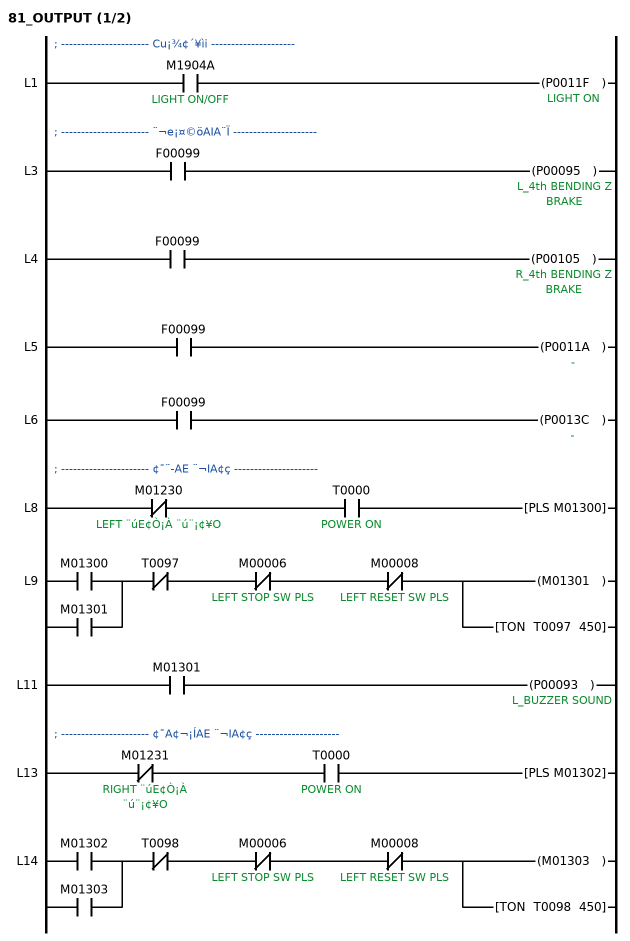
[picture p312: 81_OUTPUT rungs L1-L14]
// ---------------------- Cu¡¾¢´¥ìi ---------------------
; L1
LOAD      M1904A	// LIGHT ON/OFF
OUT       P0011F	// LIGHT ON
// ---------------------- ¨¬e¡¤©öAIA¨Ï ---------------------
; L3
LOAD      F00099
OUT       P00095	// L_4th BENDING Z BRAKE
; L4
LOAD      F00099
OUT       P00105	// R_4th BENDING Z BRAKE
; L5
LOAD      F00099
OUT       P0011A	// -
; L6
LOAD      F00099
OUT       P0013C	// -
// ---------------------- ¢¯¨­AE ¨¬IA¢ç ---------------------
; L8
LOAD NOT  M01230	// LEFT ¨úE¢Ò¡À ¨ú¨¡¢¥O
AND       T0000	// POWER ON
OUTP      M01300
; L9
LOAD      M01300
OR        M01301
AND NOT   T0097
AND NOT   M00006	// LEFT STOP SW PLS
AND NOT   M00008	// LEFT RESET SW PLS
OUT       M01301
TON       T0097 450
; L11
LOAD      M01301
OUT       P00093	// L_BUZZER SOUND
// ---------------------- ¢¯A¢¬¡ÍAE ¨¬IA¢ç ---------------------
; L13
LOAD NOT  M01231	// RIGHT ¨úE¢Ò¡À ¨ú¨¡¢¥O
AND       T0000	// POWER ON
OUTP      M01302
; L14
LOAD      M01302
OR        M01303
AND NOT   T0098
AND NOT   M00006	// LEFT STOP SW PLS
AND NOT   M00008	// LEFT RESET SW PLS
OUT       M01303
TON       T0098 450

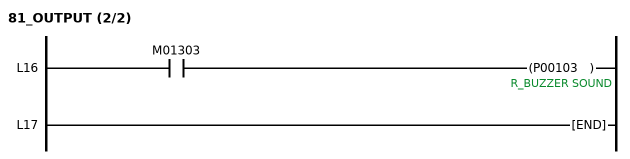
; L16
LOAD      M01303
OUT       P00103	// R_BUZZER SOUND
; L17
END

PROGRAM 82_L_MANUAL (task: ¨ö¨¬A¥ì CA¡¤I¡¾¡¿¡¤¡Í)

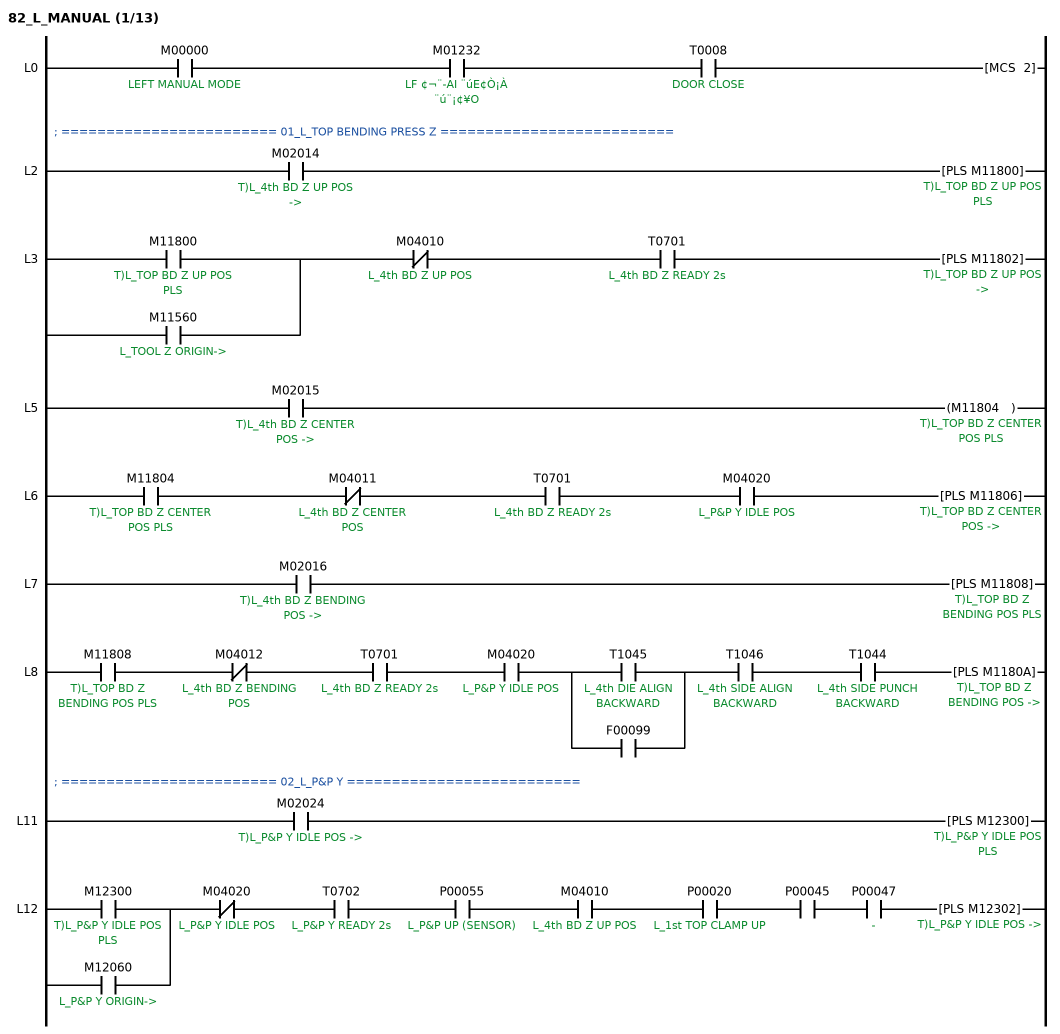
; L0
LOAD      M00000	// LEFT MANUAL MODE
AND       M01232	// LF ¢¬¨­AI ¨úE¢Ò¡À ¨ú¨¡¢¥O
AND       T0008	// DOOR CLOSE
MCS       2
// ======================== 01_L_TOP BENDING PRESS Z ==========================
; L2
LOAD      M02014	// T)L_4th BD Z UP POS ->
OUTP      M11800	// T)L_TOP BD Z UP POS PLS
; L3
LOAD      M11800	// T)L_TOP BD Z UP POS PLS
OR        M11560	// L_TOOL Z ORIGIN->
AND NOT   M04010	// L_4th BD Z UP POS
AND       T0701	// L_4th BD Z READY 2s
OUTP      M11802	// T)L_TOP BD Z UP POS ->
; L5
LOAD      M02015	// T)L_4th BD Z CENTER POS ->
OUT       M11804	// T)L_TOP BD Z CENTER POS PLS
; L6
LOAD      M11804	// T)L_TOP BD Z CENTER POS PLS
AND NOT   M04011	// L_4th BD Z CENTER POS
AND       T0701	// L_4th BD Z READY 2s
AND       M04020	// L_P&P Y IDLE POS
OUTP      M11806	// T)L_TOP BD Z CENTER POS ->
; L7
LOAD      M02016	// T)L_4th BD Z BENDING POS ->
OUTP      M11808	// T)L_TOP BD Z BENDING POS PLS
; L8
LOAD      M11808	// T)L_TOP BD Z BENDING POS PLS
AND NOT   M04012	// L_4th BD Z BENDING POS
AND       T0701	// L_4th BD Z READY 2s
AND       M04020	// L_P&P Y IDLE POS
LOAD      T1045	// L_4th DIE ALIGN BACKWARD
OR        F00099
AND LOAD
AND       T1046	// L_4th SIDE ALIGN BACKWARD
AND       T1044	// L_4th SIDE PUNCH BACKWARD
OUTP      M1180A	// T)L_TOP BD Z BENDING POS ->
// ======================== 02_L_P&P Y ==========================
; L11
LOAD      M02024	// T)L_P&P Y IDLE POS ->
OUTP      M12300	// T)L_P&P Y IDLE POS PLS
; L12
LOAD      M12300	// T)L_P&P Y IDLE POS PLS
OR        M12060	// L_P&P Y ORIGIN->
AND NOT   M04020	// L_P&P Y IDLE POS
AND       T0702	// L_P&P Y READY 2s
AND       P00055	// L_P&P UP (SENSOR)
AND       M04010	// L_4th BD Z UP POS
AND       P00020	// L_1st TOP CLAMP UP
AND       P00045
AND       P00047	// -
OUTP      M12302	// T)L_P&P Y IDLE POS ->

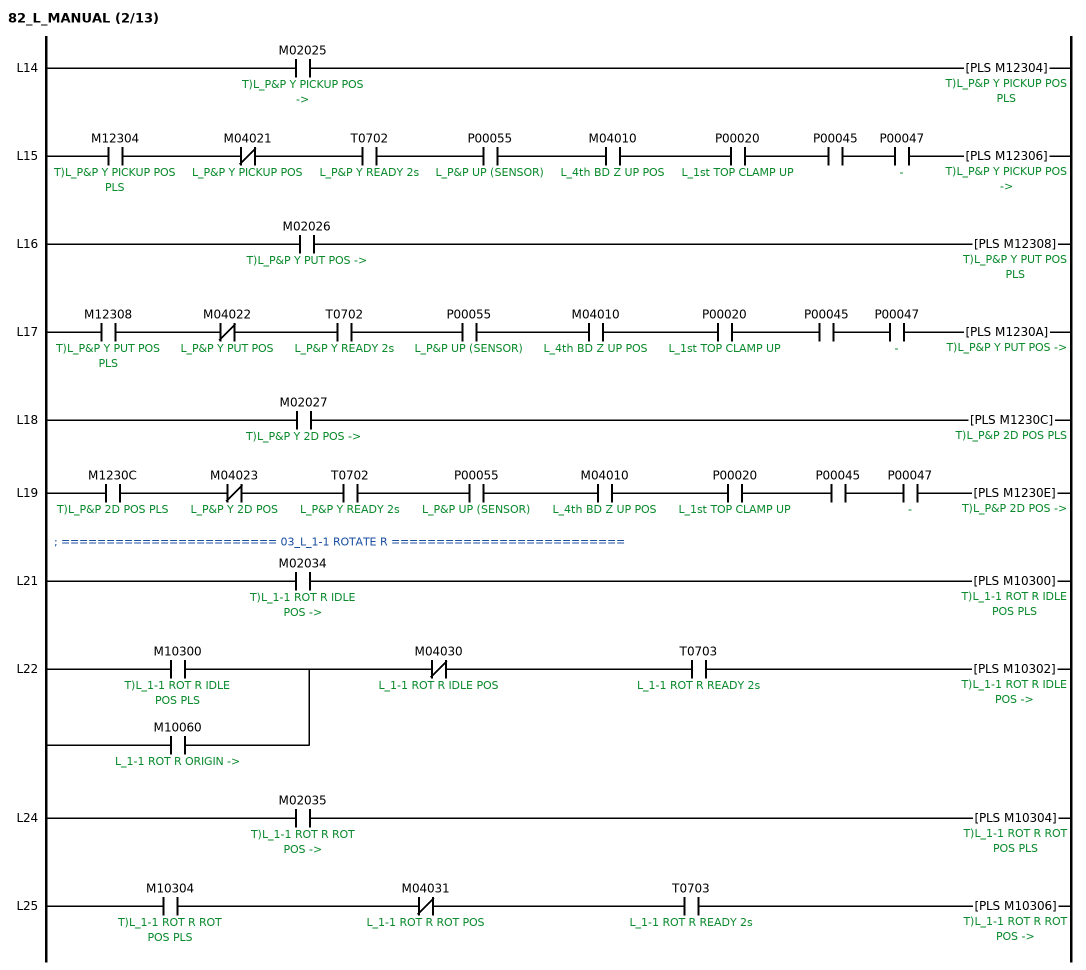
; L14
LOAD      M02025	// T)L_P&P Y PICKUP POS ->
OUTP      M12304	// T)L_P&P Y PICKUP POS PLS
; L15
LOAD      M12304	// T)L_P&P Y PICKUP POS PLS
AND NOT   M04021	// L_P&P Y PICKUP POS
AND       T0702	// L_P&P Y READY 2s
AND       P00055	// L_P&P UP (SENSOR)
AND       M04010	// L_4th BD Z UP POS
AND       P00020	// L_1st TOP CLAMP UP
AND       P00045
AND       P00047	// -
OUTP      M12306	// T)L_P&P Y PICKUP POS ->
; L16
LOAD      M02026	// T)L_P&P Y PUT POS ->
OUTP      M12308	// T)L_P&P Y PUT POS PLS
; L17
LOAD      M12308	// T)L_P&P Y PUT POS PLS
AND NOT   M04022	// L_P&P Y PUT POS
AND       T0702	// L_P&P Y READY 2s
AND       P00055	// L_P&P UP (SENSOR)
AND       M04010	// L_4th BD Z UP POS
AND       P00020	// L_1st TOP CLAMP UP
AND       P00045
AND       P00047	// -
OUTP      M1230A	// T)L_P&P Y PUT POS ->
; L18
LOAD      M02027	// T)L_P&P Y 2D POS ->
OUTP      M1230C	// T)L_P&P 2D POS PLS
; L19
LOAD      M1230C	// T)L_P&P 2D POS PLS
AND NOT   M04023	// L_P&P Y 2D POS
AND       T0702	// L_P&P Y READY 2s
AND       P00055	// L_P&P UP (SENSOR)
AND       M04010	// L_4th BD Z UP POS
AND       P00020	// L_1st TOP CLAMP UP
AND       P00045
AND       P00047	// -
OUTP      M1230E	// T)L_P&P 2D POS ->
// ======================== 03_L_1-1 ROTATE R ==========================
; L21
LOAD      M02034	// T)L_1-1 ROT R IDLE POS ->
OUTP      M10300	// T)L_1-1 ROT R IDLE POS PLS
; L22
LOAD      M10300	// T)L_1-1 ROT R IDLE POS PLS
OR        M10060	// L_1-1 ROT R ORIGIN ->
AND NOT   M04030	// L_1-1 ROT R IDLE POS
AND       T0703	// L_1-1 ROT R READY 2s
OUTP      M10302	// T)L_1-1 ROT R IDLE POS ->
; L24
LOAD      M02035	// T)L_1-1 ROT R ROT POS ->
OUTP      M10304	// T)L_1-1 ROT R ROT POS PLS
; L25
LOAD      M10304	// T)L_1-1 ROT R ROT POS PLS
AND NOT   M04031	// L_1-1 ROT R ROT POS
AND       T0703	// L_1-1 ROT R READY 2s
OUTP      M10306	// T)L_1-1 ROT R ROT POS ->

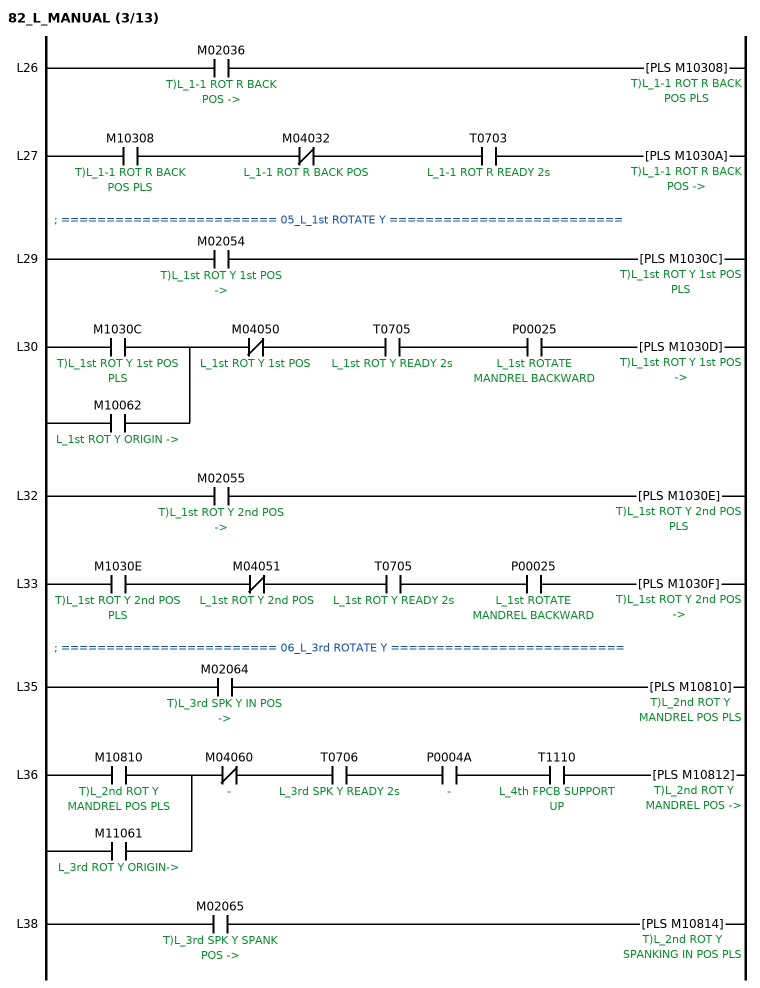
; L26
LOAD      M02036	// T)L_1-1 ROT R BACK POS ->
OUTP      M10308	// T)L_1-1 ROT R BACK POS PLS
; L27
LOAD      M10308	// T)L_1-1 ROT R BACK POS PLS
AND NOT   M04032	// L_1-1 ROT R BACK POS
AND       T0703	// L_1-1 ROT R READY 2s
OUTP      M1030A	// T)L_1-1 ROT R BACK POS ->
// ======================== 05_L_1st ROTATE Y ==========================
; L29
LOAD      M02054	// T)L_1st ROT Y 1st POS ->
OUTP      M1030C	// T)L_1st ROT Y 1st POS PLS
; L30
LOAD      M1030C	// T)L_1st ROT Y 1st POS PLS
OR        M10062	// L_1st ROT Y ORIGIN ->
AND NOT   M04050	// L_1st ROT Y 1st POS
AND       T0705	// L_1st ROT Y READY 2s
AND       P00025	// L_1st ROTATE MANDREL BACKWARD
OUTP      M1030D	// T)L_1st ROT Y 1st POS ->
; L32
LOAD      M02055	// T)L_1st ROT Y 2nd POS ->
OUTP      M1030E	// T)L_1st ROT Y 2nd POS PLS
; L33
LOAD      M1030E	// T)L_1st ROT Y 2nd POS PLS
AND NOT   M04051	// L_1st ROT Y 2nd POS
AND       T0705	// L_1st ROT Y READY 2s
AND       P00025	// L_1st ROTATE MANDREL BACKWARD
OUTP      M1030F	// T)L_1st ROT Y 2nd POS ->
// ======================== 06_L_3rd ROTATE Y ==========================
; L35
LOAD      M02064	// T)L_3rd SPK Y IN POS ->
OUTP      M10810	// T)L_2nd ROT Y MANDREL POS PLS
; L36
LOAD      M10810	// T)L_2nd ROT Y MANDREL POS PLS
OR        M11061	// L_3rd ROT Y ORIGIN->
AND NOT   M04060	// -
AND       T0706	// L_3rd SPK Y READY 2s
AND       P0004A	// -
AND       T1110	// L_4th FPCB SUPPORT UP
OUTP      M10812	// T)L_2nd ROT Y MANDREL POS ->
; L38
LOAD      M02065	// T)L_3rd SPK Y SPANK POS ->
OUTP      M10814	// T)L_2nd ROT Y SPANKING IN POS PLS

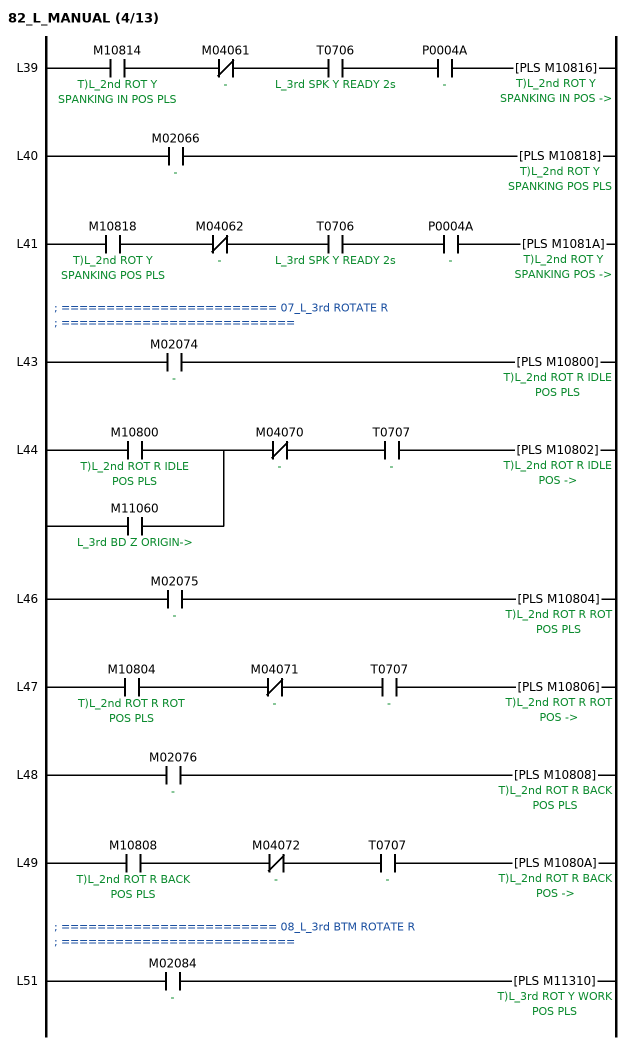
; L39
LOAD      M10814	// T)L_2nd ROT Y SPANKING IN POS PLS
AND NOT   M04061	// -
AND       T0706	// L_3rd SPK Y READY 2s
AND       P0004A	// -
OUTP      M10816	// T)L_2nd ROT Y SPANKING IN POS ->
; L40
LOAD      M02066	// -
OUTP      M10818	// T)L_2nd ROT Y SPANKING POS PLS
; L41
LOAD      M10818	// T)L_2nd ROT Y SPANKING POS PLS
AND NOT   M04062	// -
AND       T0706	// L_3rd SPK Y READY 2s
AND       P0004A	// -
OUTP      M1081A	// T)L_2nd ROT Y SPANKING POS ->
// ======================== 07_L_3rd ROTATE R ==========================
; L43
LOAD      M02074	// -
OUTP      M10800	// T)L_2nd ROT R IDLE POS PLS
; L44
LOAD      M10800	// T)L_2nd ROT R IDLE POS PLS
OR        M11060	// L_3rd BD Z ORIGIN->
AND NOT   M04070	// -
AND       T0707	// -
OUTP      M10802	// T)L_2nd ROT R IDLE POS ->
; L46
LOAD      M02075	// -
OUTP      M10804	// T)L_2nd ROT R ROT POS PLS
; L47
LOAD      M10804	// T)L_2nd ROT R ROT POS PLS
AND NOT   M04071	// -
AND       T0707	// -
OUTP      M10806	// T)L_2nd ROT R ROT POS ->
; L48
LOAD      M02076	// -
OUTP      M10808	// T)L_2nd ROT R BACK POS PLS
; L49
LOAD      M10808	// T)L_2nd ROT R BACK POS PLS
AND NOT   M04072	// -
AND       T0707	// -
OUTP      M1080A	// T)L_2nd ROT R BACK POS ->
// ======================== 08_L_3rd BTM ROTATE R ==========================
; L51
LOAD      M02084	// -
OUTP      M11310	// T)L_3rd ROT Y WORK POS PLS

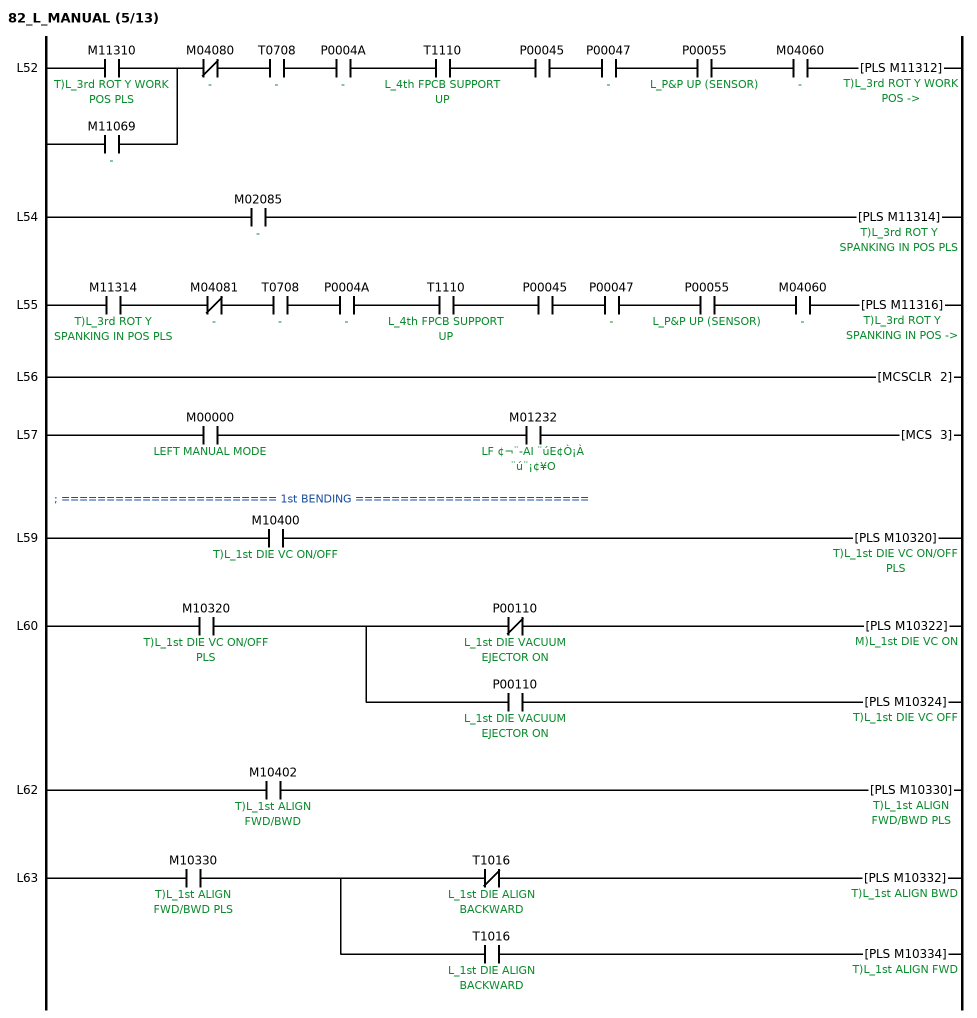
; L52
LOAD      M11310	// T)L_3rd ROT Y WORK POS PLS
OR        M11069	// -
AND NOT   M04080	// -
AND       T0708	// -
AND       P0004A	// -
AND       T1110	// L_4th FPCB SUPPORT UP
AND       P00045
AND       P00047	// -
AND       P00055	// L_P&P UP (SENSOR)
AND       M04060	// -
OUTP      M11312	// T)L_3rd ROT Y WORK POS ->
; L54
LOAD      M02085	// -
OUTP      M11314	// T)L_3rd ROT Y SPANKING IN POS PLS
; L55
LOAD      M11314	// T)L_3rd ROT Y SPANKING IN POS PLS
AND NOT   M04081	// -
AND       T0708	// -
AND       P0004A	// -
AND       T1110	// L_4th FPCB SUPPORT UP
AND       P00045
AND       P00047	// -
AND       P00055	// L_P&P UP (SENSOR)
AND       M04060	// -
OUTP      M11316	// T)L_3rd ROT Y SPANKING IN POS ->
; L56
MCSCLR    2
; L57
LOAD      M00000	// LEFT MANUAL MODE
AND       M01232	// LF ¢¬¨­AI ¨úE¢Ò¡À ¨ú¨¡¢¥O
MCS       3
// ======================== 1st BENDING ==========================
; L59
LOAD      M10400	// T)L_1st DIE VC ON/OFF
OUTP      M10320	// T)L_1st DIE VC ON/OFF PLS
; L60
LOAD      M10320	// T)L_1st DIE VC ON/OFF PLS
MPUSH
AND NOT   P00110	// L_1st DIE VACUUM EJECTOR ON
OUTP      M10322	// M)L_1st DIE VC ON
MPOP
AND       P00110	// L_1st DIE VACUUM EJECTOR ON
OUTP      M10324	// T)L_1st DIE VC OFF
; L62
LOAD      M10402	// T)L_1st ALIGN FWD/BWD
OUTP      M10330	// T)L_1st ALIGN FWD/BWD PLS
; L63
LOAD      M10330	// T)L_1st ALIGN FWD/BWD PLS
MPUSH
AND NOT   T1016	// L_1st DIE ALIGN BACKWARD
OUTP      M10332	// T)L_1st ALIGN BWD
MPOP
AND       T1016	// L_1st DIE ALIGN BACKWARD
OUTP      M10334	// T)L_1st ALIGN FWD

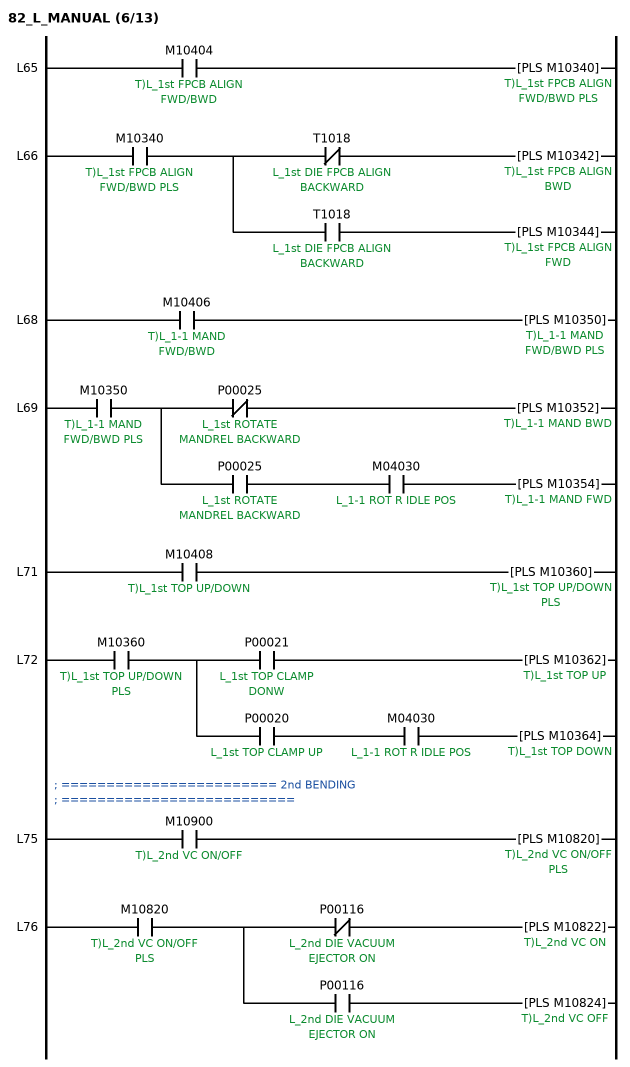
; L65
LOAD      M10404	// T)L_1st FPCB ALIGN FWD/BWD
OUTP      M10340	// T)L_1st FPCB ALIGN FWD/BWD PLS
; L66
LOAD      M10340	// T)L_1st FPCB ALIGN FWD/BWD PLS
MPUSH
AND NOT   T1018	// L_1st DIE FPCB ALIGN BACKWARD
OUTP      M10342	// T)L_1st FPCB ALIGN BWD
MPOP
AND       T1018	// L_1st DIE FPCB ALIGN BACKWARD
OUTP      M10344	// T)L_1st FPCB ALIGN FWD
; L68
LOAD      M10406	// T)L_1-1 MAND FWD/BWD
OUTP      M10350	// T)L_1-1 MAND FWD/BWD PLS
; L69
LOAD      M10350	// T)L_1-1 MAND FWD/BWD PLS
MPUSH
AND NOT   P00025	// L_1st ROTATE MANDREL BACKWARD
OUTP      M10352	// T)L_1-1 MAND BWD
MPOP
AND       P00025	// L_1st ROTATE MANDREL BACKWARD
AND       M04030	// L_1-1 ROT R IDLE POS
OUTP      M10354	// T)L_1-1 MAND FWD
; L71
LOAD      M10408	// T)L_1st TOP UP/DOWN
OUTP      M10360	// T)L_1st TOP UP/DOWN PLS
; L72
LOAD      M10360	// T)L_1st TOP UP/DOWN PLS
MPUSH
AND       P00021	// L_1st TOP CLAMP DONW
OUTP      M10362	// T)L_1st TOP UP
MPOP
AND       P00020	// L_1st TOP CLAMP UP
AND       M04030	// L_1-1 ROT R IDLE POS
OUTP      M10364	// T)L_1st TOP DOWN
// ======================== 2nd BENDING ==========================
; L75
LOAD      M10900	// T)L_2nd VC ON/OFF
OUTP      M10820	// T)L_2nd VC ON/OFF PLS
; L76
LOAD      M10820	// T)L_2nd VC ON/OFF PLS
MPUSH
AND NOT   P00116	// L_2nd DIE VACUUM EJECTOR ON
OUTP      M10822	// T)L_2nd VC ON
MPOP
AND       P00116	// L_2nd DIE VACUUM EJECTOR ON
OUTP      M10824	// T)L_2nd VC OFF

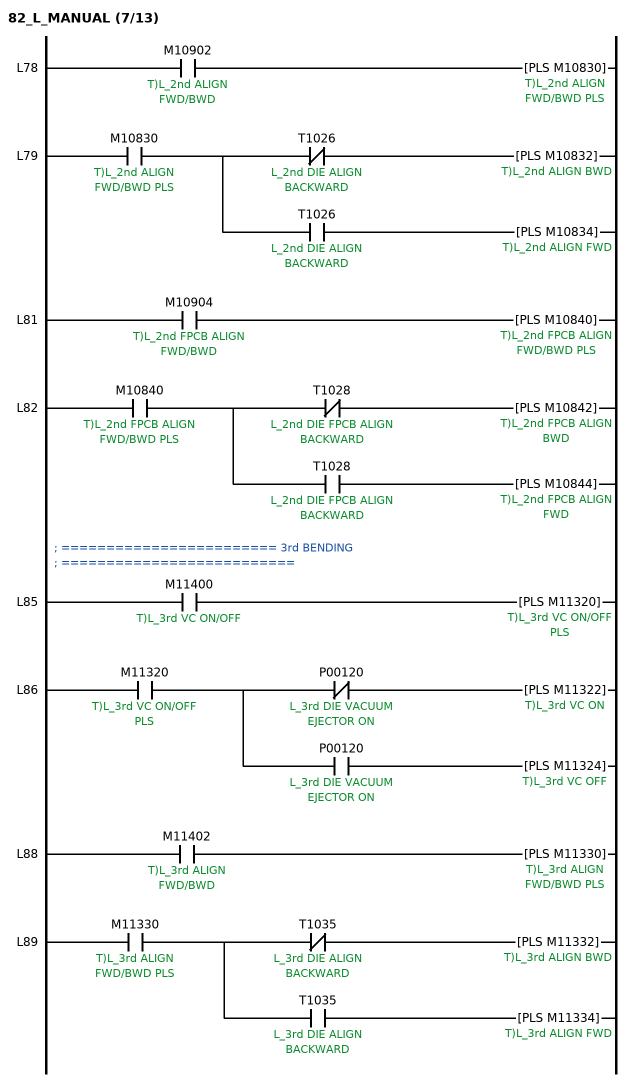
; L78
LOAD      M10902	// T)L_2nd ALIGN FWD/BWD
OUTP      M10830	// T)L_2nd ALIGN FWD/BWD PLS
; L79
LOAD      M10830	// T)L_2nd ALIGN FWD/BWD PLS
MPUSH
AND NOT   T1026	// L_2nd DIE ALIGN BACKWARD
OUTP      M10832	// T)L_2nd ALIGN BWD
MPOP
AND       T1026	// L_2nd DIE ALIGN BACKWARD
OUTP      M10834	// T)L_2nd ALIGN FWD
; L81
LOAD      M10904	// T)L_2nd FPCB ALIGN FWD/BWD
OUTP      M10840	// T)L_2nd FPCB ALIGN FWD/BWD PLS
; L82
LOAD      M10840	// T)L_2nd FPCB ALIGN FWD/BWD PLS
MPUSH
AND NOT   T1028	// L_2nd DIE FPCB ALIGN BACKWARD
OUTP      M10842	// T)L_2nd FPCB ALIGN BWD
MPOP
AND       T1028	// L_2nd DIE FPCB ALIGN BACKWARD
OUTP      M10844	// T)L_2nd FPCB ALIGN FWD
// ======================== 3rd BENDING ==========================
; L85
LOAD      M11400	// T)L_3rd VC ON/OFF
OUTP      M11320	// T)L_3rd VC ON/OFF PLS
; L86
LOAD      M11320	// T)L_3rd VC ON/OFF PLS
MPUSH
AND NOT   P00120	// L_3rd DIE VACUUM EJECTOR ON
OUTP      M11322	// T)L_3rd VC ON
MPOP
AND       P00120	// L_3rd DIE VACUUM EJECTOR ON
OUTP      M11324	// T)L_3rd VC OFF
; L88
LOAD      M11402	// T)L_3rd ALIGN FWD/BWD
OUTP      M11330	// T)L_3rd ALIGN FWD/BWD PLS
; L89
LOAD      M11330	// T)L_3rd ALIGN FWD/BWD PLS
MPUSH
AND NOT   T1035	// L_3rd DIE ALIGN BACKWARD
OUTP      M11332	// T)L_3rd ALIGN BWD
MPOP
AND       T1035	// L_3rd DIE ALIGN BACKWARD
OUTP      M11334	// T)L_3rd ALIGN FWD

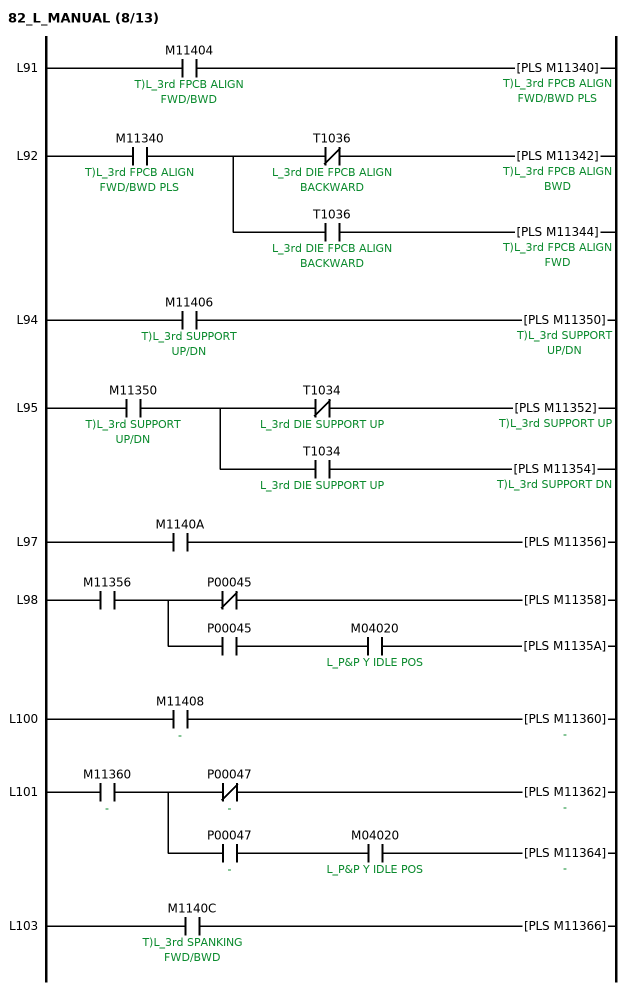
; L91
LOAD      M11404	// T)L_3rd FPCB ALIGN FWD/BWD
OUTP      M11340	// T)L_3rd FPCB ALIGN FWD/BWD PLS
; L92
LOAD      M11340	// T)L_3rd FPCB ALIGN FWD/BWD PLS
MPUSH
AND NOT   T1036	// L_3rd DIE FPCB ALIGN BACKWARD
OUTP      M11342	// T)L_3rd FPCB ALIGN BWD
MPOP
AND       T1036	// L_3rd DIE FPCB ALIGN BACKWARD
OUTP      M11344	// T)L_3rd FPCB ALIGN FWD
; L94
LOAD      M11406	// T)L_3rd SUPPORT UP/DN
OUTP      M11350	// T)L_3rd SUPPORT UP/DN
; L95
LOAD      M11350	// T)L_3rd SUPPORT UP/DN
MPUSH
AND NOT   T1034	// L_3rd DIE SUPPORT UP
OUTP      M11352	// T)L_3rd SUPPORT UP
MPOP
AND       T1034	// L_3rd DIE SUPPORT UP
OUTP      M11354	// T)L_3rd SUPPORT DN
; L97
LOAD      M1140A
OUTP      M11356
; L98
LOAD      M11356
MPUSH
AND NOT   P00045
OUTP      M11358
MPOP
AND       P00045
AND       M04020	// L_P&P Y IDLE POS
OUTP      M1135A
; L100
LOAD      M11408	// -
OUTP      M11360	// -
; L101
LOAD      M11360	// -
MPUSH
AND NOT   P00047	// -
OUTP      M11362	// -
MPOP
AND       P00047	// -
AND       M04020	// L_P&P Y IDLE POS
OUTP      M11364	// -
; L103
LOAD      M1140C	// T)L_3rd SPANKING FWD/BWD
OUTP      M11366

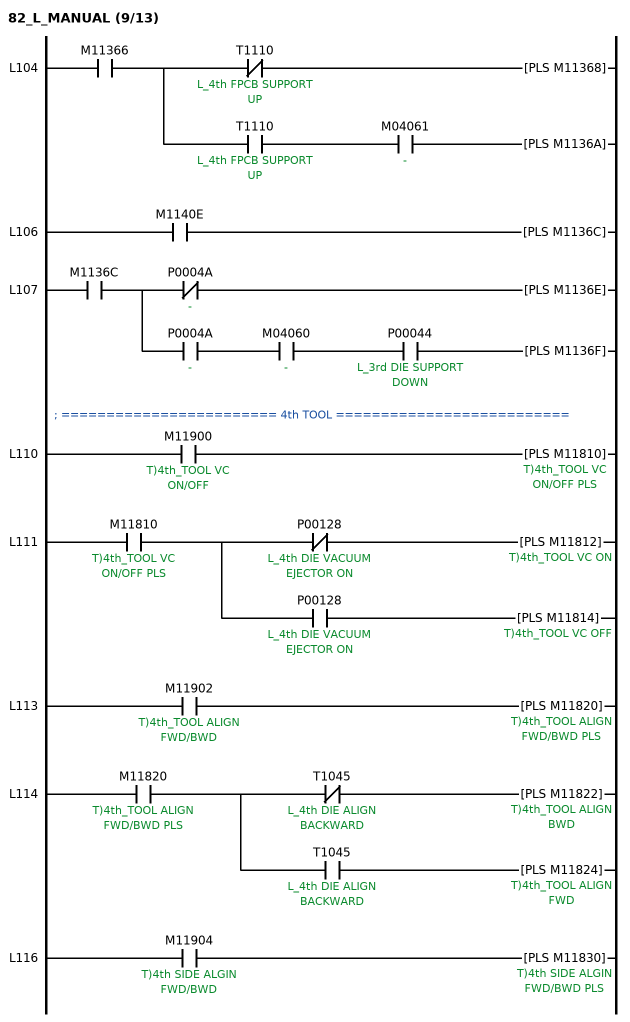
; L104
LOAD      M11366
MPUSH
AND NOT   T1110	// L_4th FPCB SUPPORT UP
OUTP      M11368
MPOP
AND       T1110	// L_4th FPCB SUPPORT UP
AND       M04061	// -
OUTP      M1136A
; L106
LOAD      M1140E
OUTP      M1136C
; L107
LOAD      M1136C
MPUSH
AND NOT   P0004A	// -
OUTP      M1136E
MPOP
AND       P0004A	// -
AND       M04060	// -
AND       P00044	// L_3rd DIE SUPPORT DOWN
OUTP      M1136F
// ======================== 4th TOOL ==========================
; L110
LOAD      M11900	// T)4th_TOOL VC ON/OFF
OUTP      M11810	// T)4th_TOOL VC ON/OFF PLS
; L111
LOAD      M11810	// T)4th_TOOL VC ON/OFF PLS
MPUSH
AND NOT   P00128	// L_4th DIE VACUUM EJECTOR ON
OUTP      M11812	// T)4th_TOOL VC ON
MPOP
AND       P00128	// L_4th DIE VACUUM EJECTOR ON
OUTP      M11814	// T)4th_TOOL VC OFF
; L113
LOAD      M11902	// T)4th_TOOL ALIGN FWD/BWD
OUTP      M11820	// T)4th_TOOL ALIGN FWD/BWD PLS
; L114
LOAD      M11820	// T)4th_TOOL ALIGN FWD/BWD PLS
MPUSH
AND NOT   T1045	// L_4th DIE ALIGN BACKWARD
OUTP      M11822	// T)4th_TOOL ALIGN BWD
MPOP
AND       T1045	// L_4th DIE ALIGN BACKWARD
OUTP      M11824	// T)4th_TOOL ALIGN FWD
; L116
LOAD      M11904	// T)4th SIDE ALGIN FWD/BWD
OUTP      M11830	// T)4th SIDE ALGIN FWD/BWD PLS

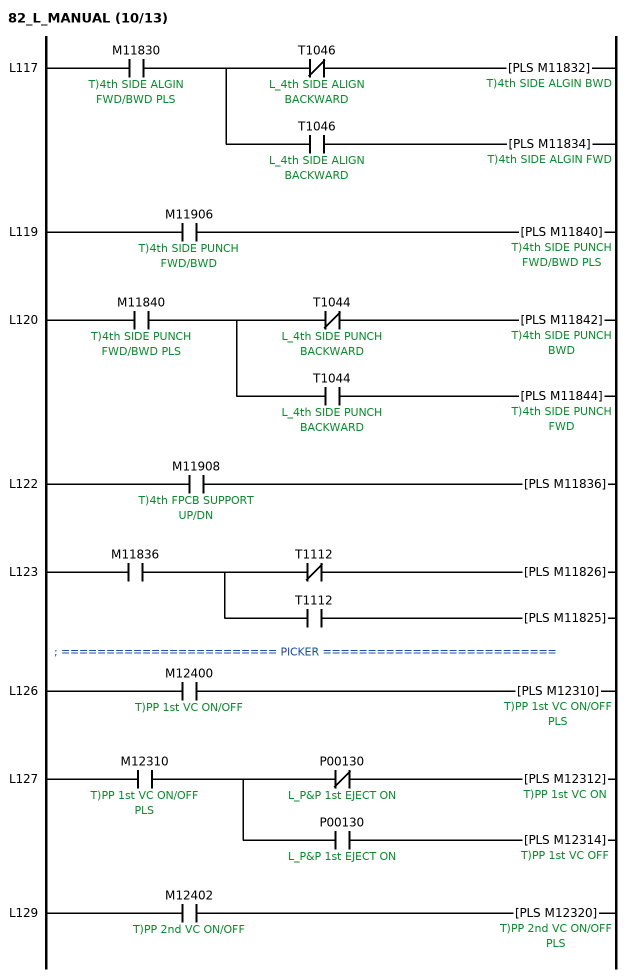
; L117
LOAD      M11830	// T)4th SIDE ALGIN FWD/BWD PLS
MPUSH
AND NOT   T1046	// L_4th SIDE ALIGN BACKWARD
OUTP      M11832	// T)4th SIDE ALGIN BWD
MPOP
AND       T1046	// L_4th SIDE ALIGN BACKWARD
OUTP      M11834	// T)4th SIDE ALGIN FWD
; L119
LOAD      M11906	// T)4th SIDE PUNCH FWD/BWD
OUTP      M11840	// T)4th SIDE PUNCH FWD/BWD PLS
; L120
LOAD      M11840	// T)4th SIDE PUNCH FWD/BWD PLS
MPUSH
AND NOT   T1044	// L_4th SIDE PUNCH BACKWARD
OUTP      M11842	// T)4th SIDE PUNCH BWD
MPOP
AND       T1044	// L_4th SIDE PUNCH BACKWARD
OUTP      M11844	// T)4th SIDE PUNCH FWD
; L122
LOAD      M11908	// T)4th FPCB SUPPORT UP/DN
OUTP      M11836
; L123
LOAD      M11836
MPUSH
AND NOT   T1112
OUTP      M11826
MPOP
AND       T1112
OUTP      M11825
// ======================== PICKER ==========================
; L126
LOAD      M12400	// T)PP 1st VC ON/OFF
OUTP      M12310	// T)PP 1st VC ON/OFF PLS
; L127
LOAD      M12310	// T)PP 1st VC ON/OFF PLS
MPUSH
AND NOT   P00130	// L_P&P 1st EJECT ON
OUTP      M12312	// T)PP 1st VC ON
MPOP
AND       P00130	// L_P&P 1st EJECT ON
OUTP      M12314	// T)PP 1st VC OFF
; L129
LOAD      M12402	// T)PP 2nd VC ON/OFF
OUTP      M12320	// T)PP 2nd VC ON/OFF PLS

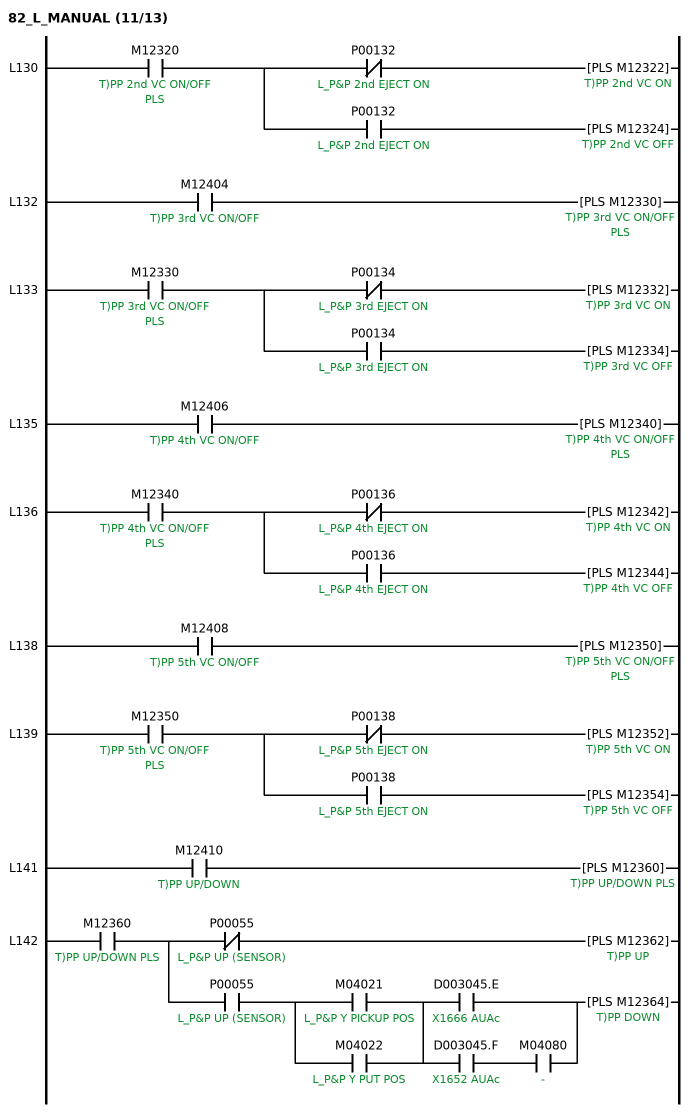
; L130
LOAD      M12320	// T)PP 2nd VC ON/OFF PLS
MPUSH
AND NOT   P00132	// L_P&P 2nd EJECT ON
OUTP      M12322	// T)PP 2nd VC ON
MPOP
AND       P00132	// L_P&P 2nd EJECT ON
OUTP      M12324	// T)PP 2nd VC OFF
; L132
LOAD      M12404	// T)PP 3rd VC ON/OFF
OUTP      M12330	// T)PP 3rd VC ON/OFF PLS
; L133
LOAD      M12330	// T)PP 3rd VC ON/OFF PLS
MPUSH
AND NOT   P00134	// L_P&P 3rd EJECT ON
OUTP      M12332	// T)PP 3rd VC ON
MPOP
AND       P00134	// L_P&P 3rd EJECT ON
OUTP      M12334	// T)PP 3rd VC OFF
; L135
LOAD      M12406	// T)PP 4th VC ON/OFF
OUTP      M12340	// T)PP 4th VC ON/OFF PLS
; L136
LOAD      M12340	// T)PP 4th VC ON/OFF PLS
MPUSH
AND NOT   P00136	// L_P&P 4th EJECT ON
OUTP      M12342	// T)PP 4th VC ON
MPOP
AND       P00136	// L_P&P 4th EJECT ON
OUTP      M12344	// T)PP 4th VC OFF
; L138
LOAD      M12408	// T)PP 5th VC ON/OFF
OUTP      M12350	// T)PP 5th VC ON/OFF PLS
; L139
LOAD      M12350	// T)PP 5th VC ON/OFF PLS
MPUSH
AND NOT   P00138	// L_P&P 5th EJECT ON
OUTP      M12352	// T)PP 5th VC ON
MPOP
AND       P00138	// L_P&P 5th EJECT ON
OUTP      M12354	// T)PP 5th VC OFF
; L141
LOAD      M12410	// T)PP UP/DOWN
OUTP      M12360	// T)PP UP/DOWN PLS
; L142
LOAD      M12360	// T)PP UP/DOWN PLS
MPUSH
AND NOT   P00055	// L_P&P UP (SENSOR)
OUTP      M12362	// T)PP UP
MPOP
AND       P00055	// L_P&P UP (SENSOR)
LOAD      M04021	// L_P&P Y PICKUP POS
OR        M04022	// L_P&P Y PUT POS
AND LOAD
LOAD      D003045.E	// X1666 AUAc
LOAD      D003045.F	// X1652 AUAc
AND       M04080	// -
OR LOAD
AND LOAD
OUTP      M12364	// T)PP DOWN

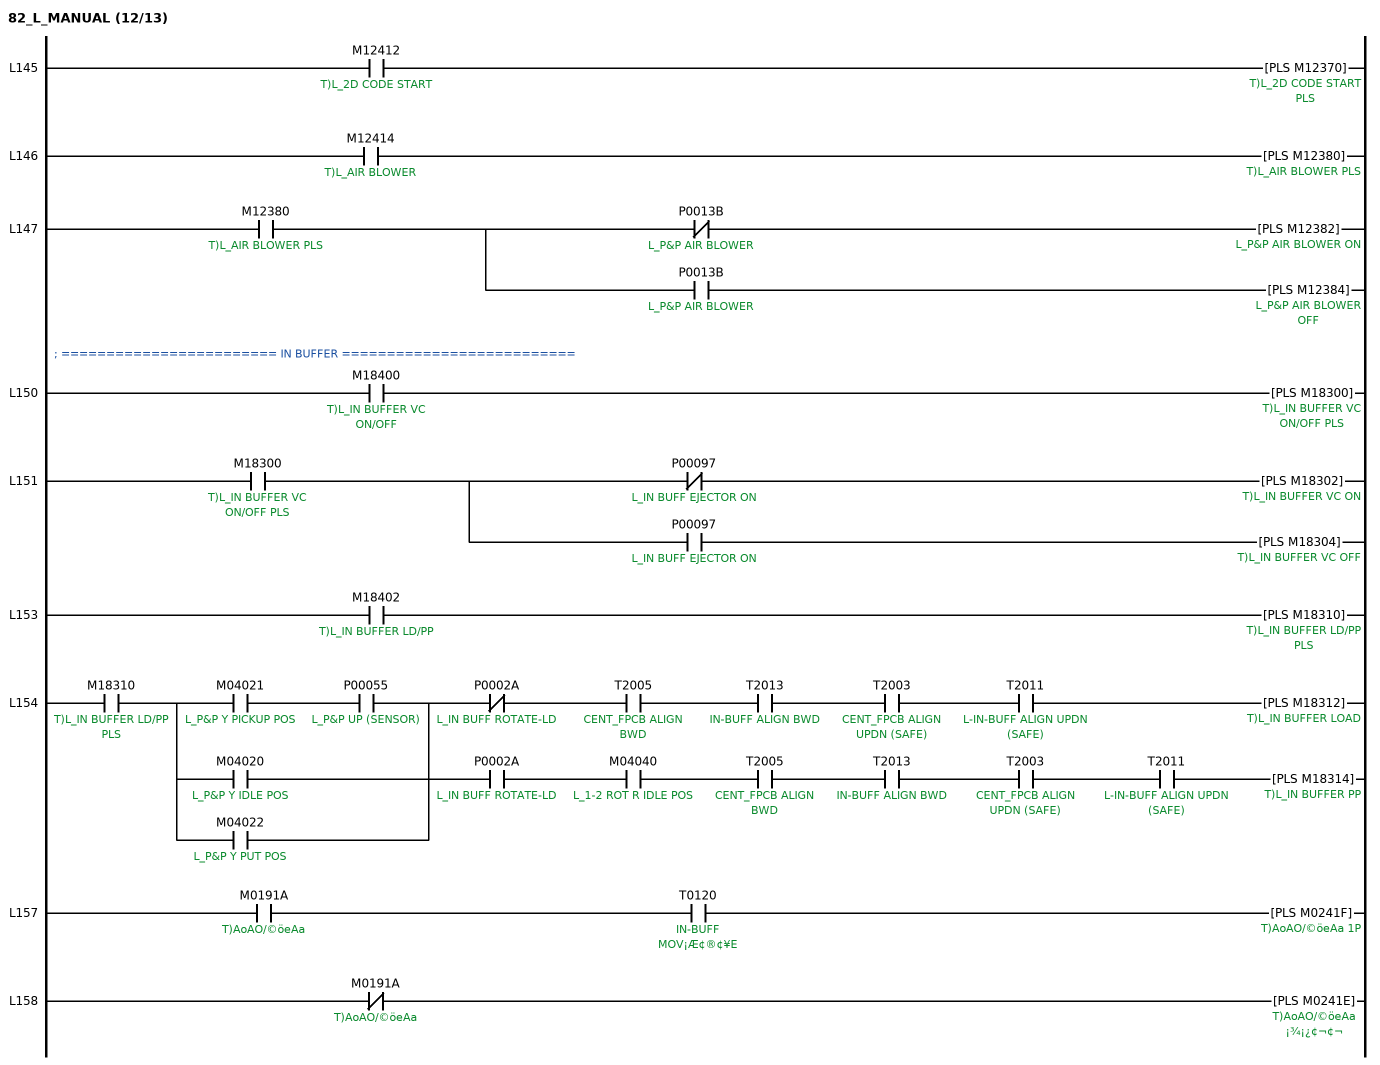
; L145
LOAD      M12412	// T)L_2D CODE START
OUTP      M12370	// T)L_2D CODE START PLS
; L146
LOAD      M12414	// T)L_AIR BLOWER
OUTP      M12380	// T)L_AIR BLOWER PLS
; L147
LOAD      M12380	// T)L_AIR BLOWER PLS
MPUSH
AND NOT   P0013B	// L_P&P AIR BLOWER
OUTP      M12382	// L_P&P AIR BLOWER ON
MPOP
AND       P0013B	// L_P&P AIR BLOWER
OUTP      M12384	// L_P&P AIR BLOWER OFF
// ======================== IN BUFFER ==========================
; L150
LOAD      M18400	// T)L_IN BUFFER VC ON/OFF
OUTP      M18300	// T)L_IN BUFFER VC ON/OFF PLS
; L151
LOAD      M18300	// T)L_IN BUFFER VC ON/OFF PLS
MPUSH
AND NOT   P00097	// L_IN BUFF EJECTOR ON
OUTP      M18302	// T)L_IN BUFFER VC ON
MPOP
AND       P00097	// L_IN BUFF EJECTOR ON
OUTP      M18304	// T)L_IN BUFFER VC OFF
; L153
LOAD      M18402	// T)L_IN BUFFER LD/PP
OUTP      M18310	// T)L_IN BUFFER LD/PP PLS
; L154
LOAD      M18310	// T)L_IN BUFFER LD/PP PLS
LOAD      M04021	// L_P&P Y PICKUP POS
AND       P00055	// L_P&P UP (SENSOR)
OR        M04020	// L_P&P Y IDLE POS
OR        M04022	// L_P&P Y PUT POS
AND LOAD
MPUSH
AND NOT   P0002A	// L_IN BUFF ROTATE-LD
AND       T2005	// CENT_FPCB ALIGN BWD
AND       T2013	// IN-BUFF ALIGN BWD
AND       T2003	// CENT_FPCB ALIGN UPDN (SAFE)
AND       T2011	// L-IN-BUFF ALIGN UPDN (SAFE)
OUTP      M18312	// T)L_IN BUFFER LOAD
MPOP
AND       P0002A	// L_IN BUFF ROTATE-LD
AND       M04040	// L_1-2 ROT R IDLE POS
AND       T2005	// CENT_FPCB ALIGN BWD
AND       T2013	// IN-BUFF ALIGN BWD
AND       T2003	// CENT_FPCB ALIGN UPDN (SAFE)
AND       T2011	// L-IN-BUFF ALIGN UPDN (SAFE)
OUTP      M18314	// T)L_IN BUFFER PP
; L157
LOAD      M0191A	// T)AoAO/©öeAa
AND       T0120	// IN-BUFF MOV¡Æ¢®¢¥E
OUTP      M0241F	// T)AoAO/©öeAa 1P
; L158
LOAD NOT  M0191A	// T)AoAO/©öeAa
OUTP      M0241E	// T)AoAO/©öeAa ¡¾¡¿¢¬¢¬

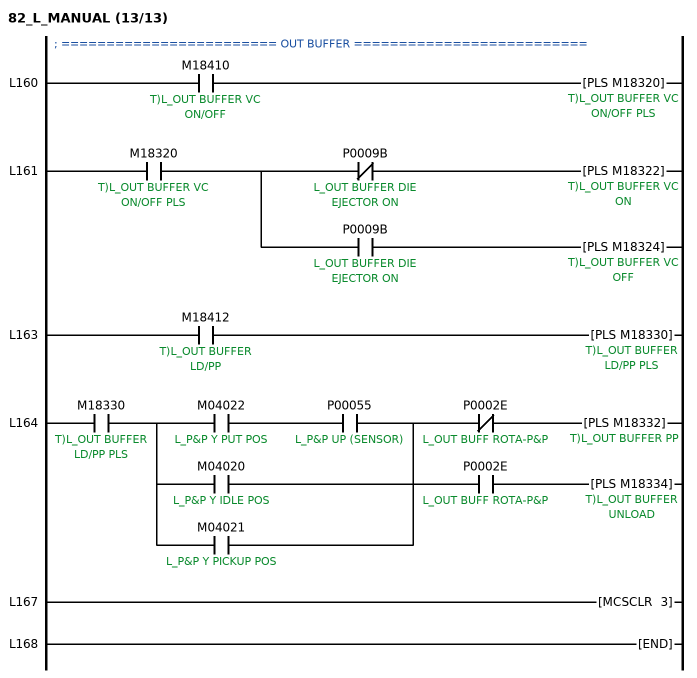
// ======================== OUT BUFFER ==========================
; L160
LOAD      M18410	// T)L_OUT BUFFER VC ON/OFF
OUTP      M18320	// T)L_OUT BUFFER VC ON/OFF PLS
; L161
LOAD      M18320	// T)L_OUT BUFFER VC ON/OFF PLS
MPUSH
AND NOT   P0009B	// L_OUT BUFFER DIE EJECTOR ON
OUTP      M18322	// T)L_OUT BUFFER VC ON
MPOP
AND       P0009B	// L_OUT BUFFER DIE EJECTOR ON
OUTP      M18324	// T)L_OUT BUFFER VC OFF
; L163
LOAD      M18412	// T)L_OUT BUFFER LD/PP
OUTP      M18330	// T)L_OUT BUFFER LD/PP PLS
; L164
LOAD      M18330	// T)L_OUT BUFFER LD/PP PLS
LOAD      M04022	// L_P&P Y PUT POS
AND       P00055	// L_P&P UP (SENSOR)
OR        M04020	// L_P&P Y IDLE POS
OR        M04021	// L_P&P Y PICKUP POS
AND LOAD
MPUSH
AND NOT   P0002E	// L_OUT BUFF ROTA-P&P
OUTP      M18332	// T)L_OUT BUFFER PP
MPOP
AND       P0002E	// L_OUT BUFF ROTA-P&P
OUTP      M18334	// T)L_OUT BUFFER UNLOAD
; L167
MCSCLR    3
; L168
END

PROGRAM 83_R_MANUAL (task: ¨ö¨¬A¥ì CA¡¤I¡¾¡¿¡¤¡Í)

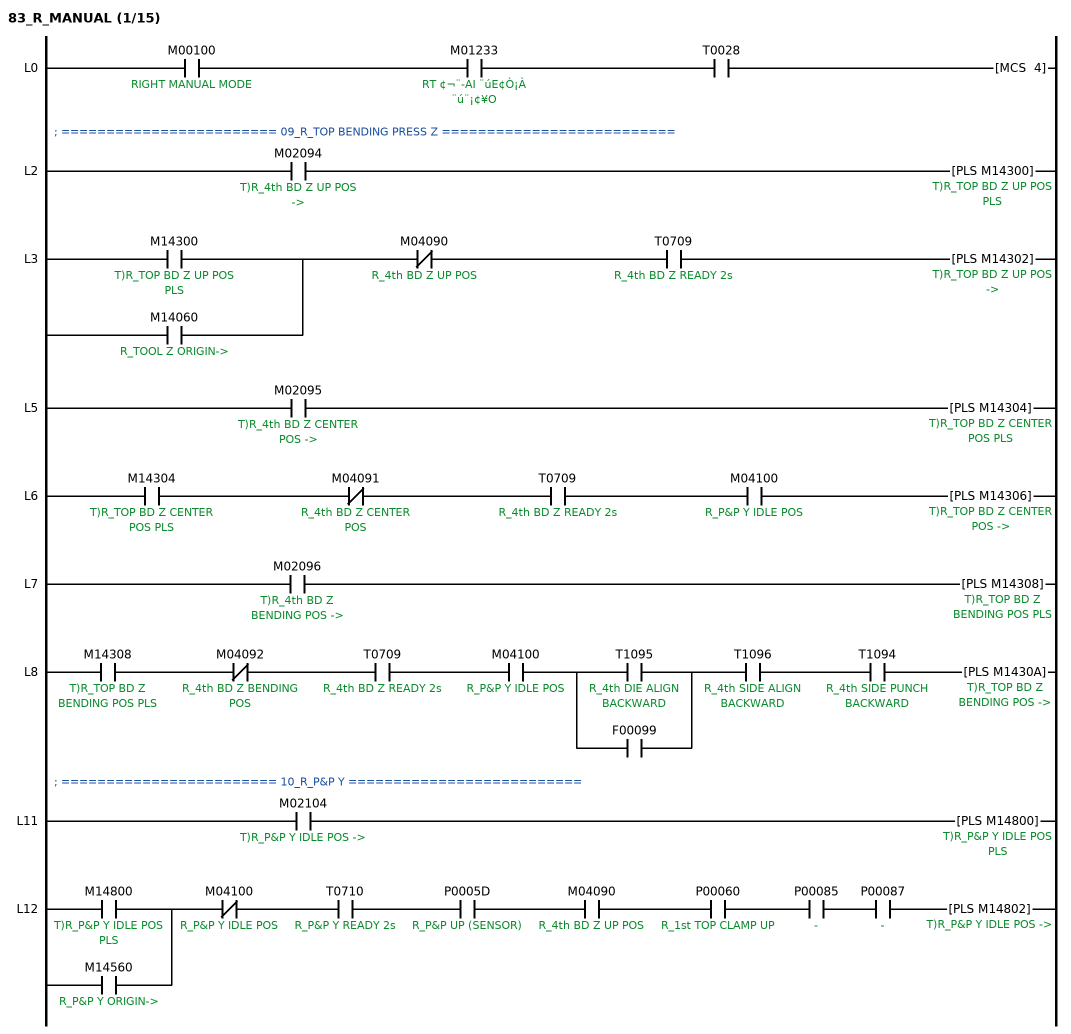
; L0
LOAD      M00100	// RIGHT MANUAL MODE
AND       M01233	// RT ¢¬¨­AI ¨úE¢Ò¡À ¨ú¨¡¢¥O
AND       T0028
MCS       4
// ======================== 09_R_TOP BENDING PRESS Z ==========================
; L2
LOAD      M02094	// T)R_4th BD Z UP POS ->
OUTP      M14300	// T)R_TOP BD Z UP POS PLS
; L3
LOAD      M14300	// T)R_TOP BD Z UP POS PLS
OR        M14060	// R_TOOL Z ORIGIN->
AND NOT   M04090	// R_4th BD Z UP POS
AND       T0709	// R_4th BD Z READY 2s
OUTP      M14302	// T)R_TOP BD Z UP POS ->
; L5
LOAD      M02095	// T)R_4th BD Z CENTER POS ->
OUTP      M14304	// T)R_TOP BD Z CENTER POS PLS
; L6
LOAD      M14304	// T)R_TOP BD Z CENTER POS PLS
AND NOT   M04091	// R_4th BD Z CENTER POS
AND       T0709	// R_4th BD Z READY 2s
AND       M04100	// R_P&P Y IDLE POS
OUTP      M14306	// T)R_TOP BD Z CENTER POS ->
; L7
LOAD      M02096	// T)R_4th BD Z BENDING POS ->
OUTP      M14308	// T)R_TOP BD Z BENDING POS PLS
; L8
LOAD      M14308	// T)R_TOP BD Z BENDING POS PLS
AND NOT   M04092	// R_4th BD Z BENDING POS
AND       T0709	// R_4th BD Z READY 2s
AND       M04100	// R_P&P Y IDLE POS
LOAD      T1095	// R_4th DIE ALIGN BACKWARD
OR        F00099
AND LOAD
AND       T1096	// R_4th SIDE ALIGN BACKWARD
AND       T1094	// R_4th SIDE PUNCH BACKWARD
OUTP      M1430A	// T)R_TOP BD Z BENDING POS ->
// ======================== 10_R_P&P Y ==========================
; L11
LOAD      M02104	// T)R_P&P Y IDLE POS ->
OUTP      M14800	// T)R_P&P Y IDLE POS PLS
; L12
LOAD      M14800	// T)R_P&P Y IDLE POS PLS
OR        M14560	// R_P&P Y ORIGIN->
AND NOT   M04100	// R_P&P Y IDLE POS
AND       T0710	// R_P&P Y READY 2s
AND       P0005D	// R_P&P UP (SENSOR)
AND       M04090	// R_4th BD Z UP POS
AND       P00060	// R_1st TOP CLAMP UP
AND       P00085	// -
AND       P00087	// -
OUTP      M14802	// T)R_P&P Y IDLE POS ->

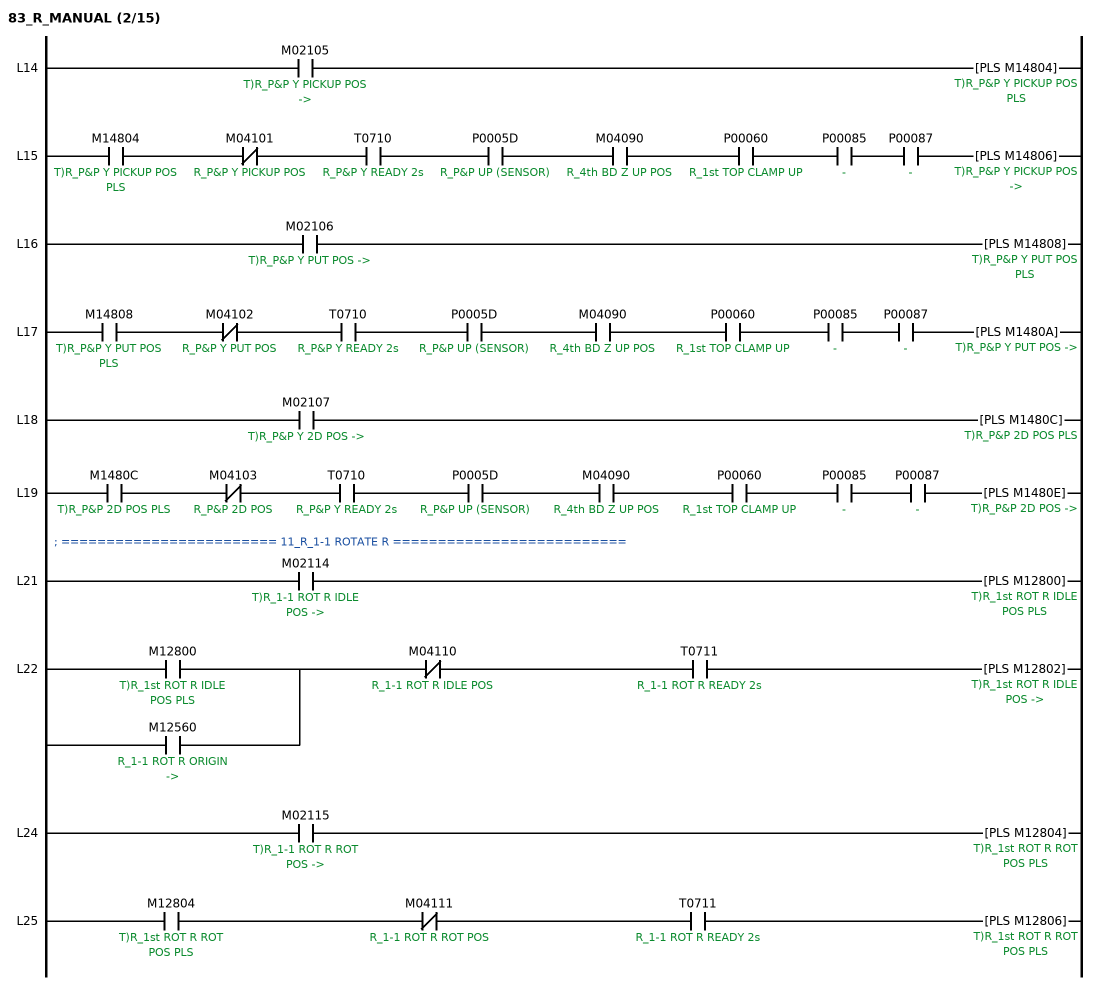
; L14
LOAD      M02105	// T)R_P&P Y PICKUP POS ->
OUTP      M14804	// T)R_P&P Y PICKUP POS PLS
; L15
LOAD      M14804	// T)R_P&P Y PICKUP POS PLS
AND NOT   M04101	// R_P&P Y PICKUP POS
AND       T0710	// R_P&P Y READY 2s
AND       P0005D	// R_P&P UP (SENSOR)
AND       M04090	// R_4th BD Z UP POS
AND       P00060	// R_1st TOP CLAMP UP
AND       P00085	// -
AND       P00087	// -
OUTP      M14806	// T)R_P&P Y PICKUP POS ->
; L16
LOAD      M02106	// T)R_P&P Y PUT POS ->
OUTP      M14808	// T)R_P&P Y PUT POS PLS
; L17
LOAD      M14808	// T)R_P&P Y PUT POS PLS
AND NOT   M04102	// R_P&P Y PUT POS
AND       T0710	// R_P&P Y READY 2s
AND       P0005D	// R_P&P UP (SENSOR)
AND       M04090	// R_4th BD Z UP POS
AND       P00060	// R_1st TOP CLAMP UP
AND       P00085	// -
AND       P00087	// -
OUTP      M1480A	// T)R_P&P Y PUT POS ->
; L18
LOAD      M02107	// T)R_P&P Y 2D POS ->
OUTP      M1480C	// T)R_P&P 2D POS PLS
; L19
LOAD      M1480C	// T)R_P&P 2D POS PLS
AND NOT   M04103	// R_P&P 2D POS
AND       T0710	// R_P&P Y READY 2s
AND       P0005D	// R_P&P UP (SENSOR)
AND       M04090	// R_4th BD Z UP POS
AND       P00060	// R_1st TOP CLAMP UP
AND       P00085	// -
AND       P00087	// -
OUTP      M1480E	// T)R_P&P 2D POS ->
// ======================== 11_R_1-1 ROTATE R ==========================
; L21
LOAD      M02114	// T)R_1-1 ROT R IDLE POS ->
OUTP      M12800	// T)R_1st ROT R IDLE POS PLS
; L22
LOAD      M12800	// T)R_1st ROT R IDLE POS PLS
OR        M12560	// R_1-1 ROT R ORIGIN ->
AND NOT   M04110	// R_1-1 ROT R IDLE POS
AND       T0711	// R_1-1 ROT R READY 2s
OUTP      M12802	// T)R_1st ROT R IDLE POS ->
; L24
LOAD      M02115	// T)R_1-1 ROT R ROT POS ->
OUTP      M12804	// T)R_1st ROT R ROT POS PLS
; L25
LOAD      M12804	// T)R_1st ROT R ROT POS PLS
AND NOT   M04111	// R_1-1 ROT R ROT POS
AND       T0711	// R_1-1 ROT R READY 2s
OUTP      M12806	// T)R_1st ROT R ROT POS PLS

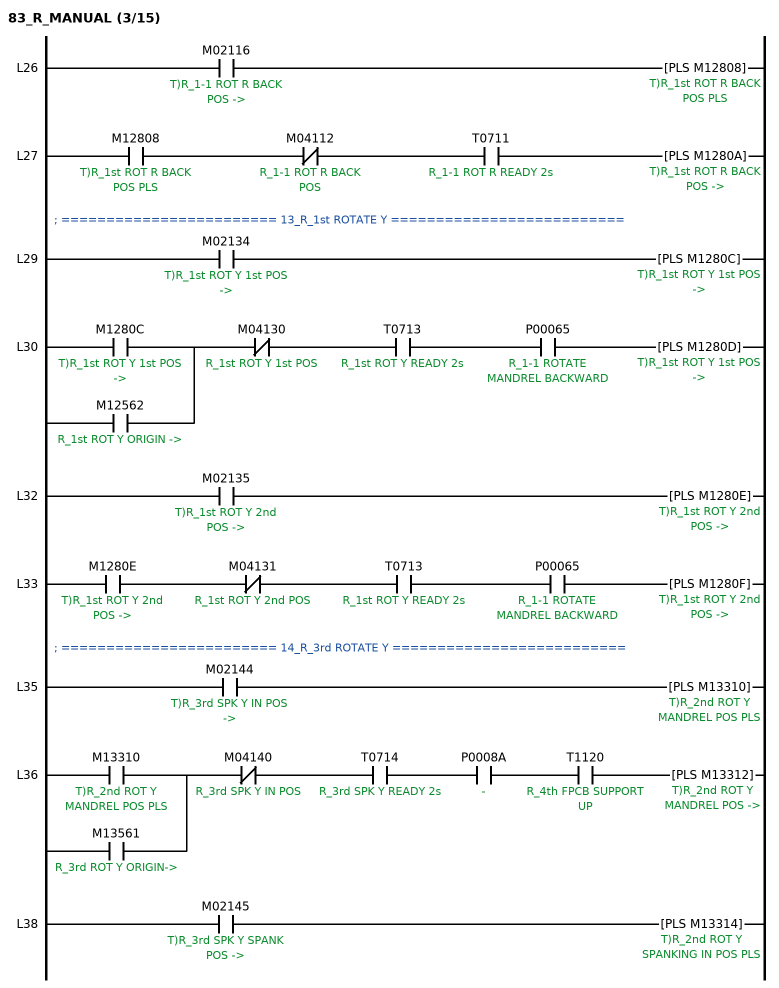
; L26
LOAD      M02116	// T)R_1-1 ROT R BACK POS ->
OUTP      M12808	// T)R_1st ROT R BACK POS PLS
; L27
LOAD      M12808	// T)R_1st ROT R BACK POS PLS
AND NOT   M04112	// R_1-1 ROT R BACK POS
AND       T0711	// R_1-1 ROT R READY 2s
OUTP      M1280A	// T)R_1st ROT R BACK POS ->
// ======================== 13_R_1st ROTATE Y ==========================
; L29
LOAD      M02134	// T)R_1st ROT Y 1st POS ->
OUTP      M1280C	// T)R_1st ROT Y 1st POS ->
; L30
LOAD      M1280C	// T)R_1st ROT Y 1st POS ->
OR        M12562	// R_1st ROT Y ORIGIN ->
AND NOT   M04130	// R_1st ROT Y 1st POS
AND       T0713	// R_1st ROT Y READY 2s
AND       P00065	// R_1-1 ROTATE MANDREL BACKWARD
OUTP      M1280D	// T)R_1st ROT Y 1st POS ->
; L32
LOAD      M02135	// T)R_1st ROT Y 2nd POS ->
OUTP      M1280E	// T)R_1st ROT Y 2nd POS ->
; L33
LOAD      M1280E	// T)R_1st ROT Y 2nd POS ->
AND NOT   M04131	// R_1st ROT Y 2nd POS
AND       T0713	// R_1st ROT Y READY 2s
AND       P00065	// R_1-1 ROTATE MANDREL BACKWARD
OUTP      M1280F	// T)R_1st ROT Y 2nd POS ->
// ======================== 14_R_3rd ROTATE Y ==========================
; L35
LOAD      M02144	// T)R_3rd SPK Y IN POS ->
OUTP      M13310	// T)R_2nd ROT Y MANDREL POS PLS
; L36
LOAD      M13310	// T)R_2nd ROT Y MANDREL POS PLS
OR        M13561	// R_3rd ROT Y ORIGIN->
AND NOT   M04140	// R_3rd SPK Y IN POS
AND       T0714	// R_3rd SPK Y READY 2s
AND       P0008A	// -
AND       T1120	// R_4th FPCB SUPPORT UP
OUTP      M13312	// T)R_2nd ROT Y MANDREL POS ->
; L38
LOAD      M02145	// T)R_3rd SPK Y SPANK POS ->
OUTP      M13314	// T)R_2nd ROT Y SPANKING IN POS PLS

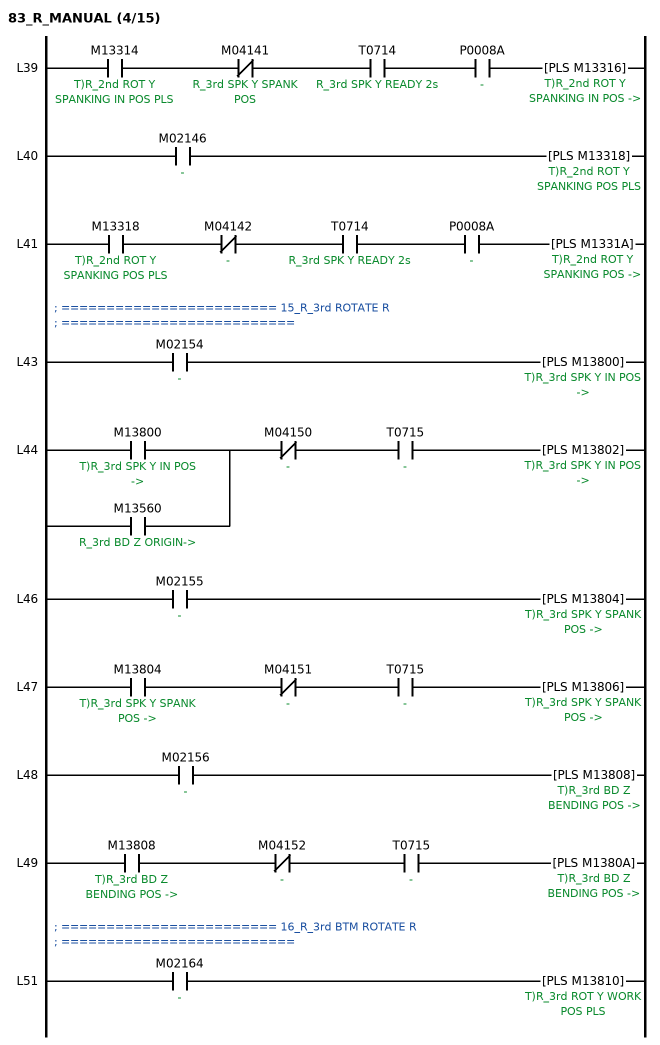
; L39
LOAD      M13314	// T)R_2nd ROT Y SPANKING IN POS PLS
AND NOT   M04141	// R_3rd SPK Y SPANK POS
AND       T0714	// R_3rd SPK Y READY 2s
AND       P0008A	// -
OUTP      M13316	// T)R_2nd ROT Y SPANKING IN POS ->
; L40
LOAD      M02146	// -
OUTP      M13318	// T)R_2nd ROT Y SPANKING POS PLS
; L41
LOAD      M13318	// T)R_2nd ROT Y SPANKING POS PLS
AND NOT   M04142	// -
AND       T0714	// R_3rd SPK Y READY 2s
AND       P0008A	// -
OUTP      M1331A	// T)R_2nd ROT Y SPANKING POS ->
// ======================== 15_R_3rd ROTATE R ==========================
; L43
LOAD      M02154	// -
OUTP      M13800	// T)R_3rd SPK Y IN POS ->
; L44
LOAD      M13800	// T)R_3rd SPK Y IN POS ->
OR        M13560	// R_3rd BD Z ORIGIN->
AND NOT   M04150	// -
AND       T0715	// -
OUTP      M13802	// T)R_3rd SPK Y IN POS ->
; L46
LOAD      M02155	// -
OUTP      M13804	// T)R_3rd SPK Y SPANK POS ->
; L47
LOAD      M13804	// T)R_3rd SPK Y SPANK POS ->
AND NOT   M04151	// -
AND       T0715	// -
OUTP      M13806	// T)R_3rd SPK Y SPANK POS ->
; L48
LOAD      M02156	// -
OUTP      M13808	// T)R_3rd BD Z BENDING POS ->
; L49
LOAD      M13808	// T)R_3rd BD Z BENDING POS ->
AND NOT   M04152	// -
AND       T0715	// -
OUTP      M1380A	// T)R_3rd BD Z BENDING POS ->
// ======================== 16_R_3rd BTM ROTATE R ==========================
; L51
LOAD      M02164	// -
OUTP      M13810	// T)R_3rd ROT Y WORK POS PLS

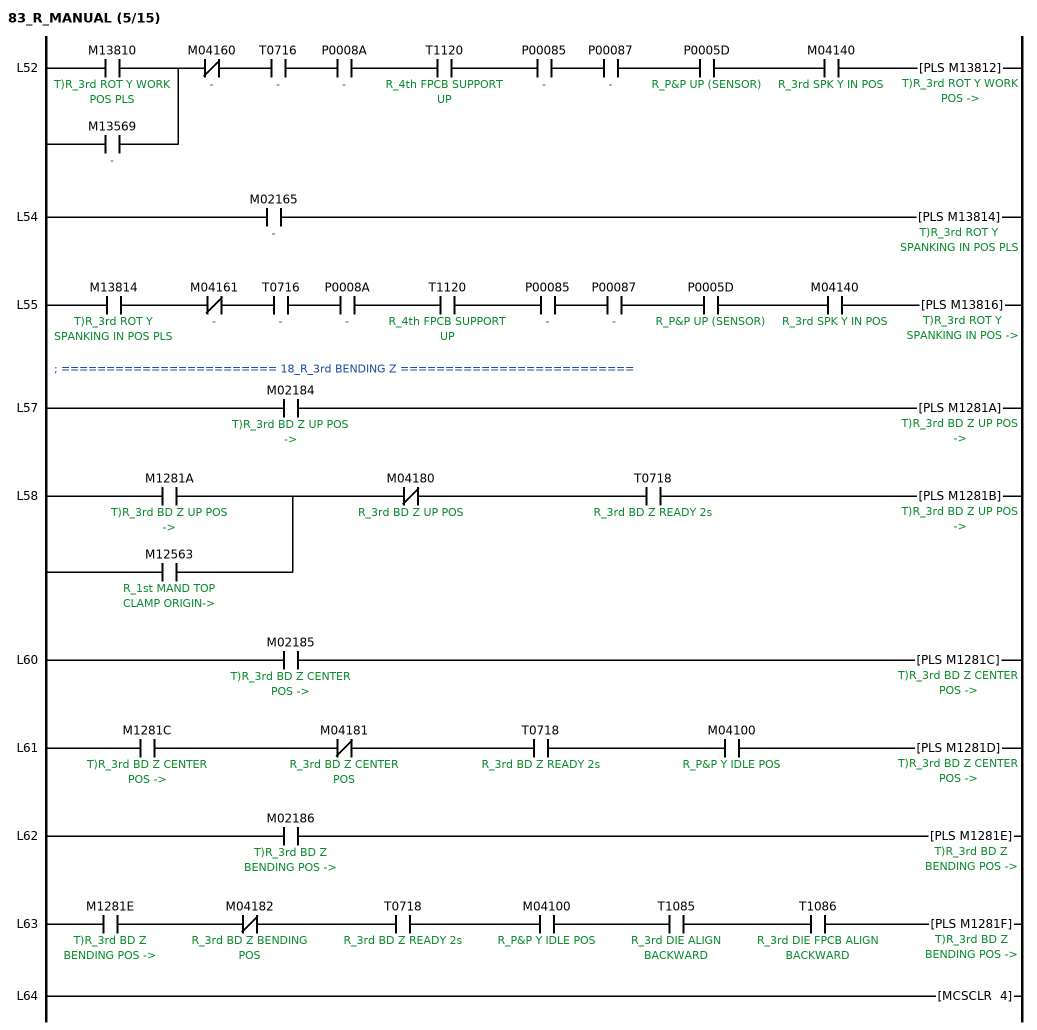
; L52
LOAD      M13810	// T)R_3rd ROT Y WORK POS PLS
OR        M13569	// -
AND NOT   M04160	// -
AND       T0716	// -
AND       P0008A	// -
AND       T1120	// R_4th FPCB SUPPORT UP
AND       P00085	// -
AND       P00087	// -
AND       P0005D	// R_P&P UP (SENSOR)
AND       M04140	// R_3rd SPK Y IN POS
OUTP      M13812	// T)R_3rd ROT Y WORK POS ->
; L54
LOAD      M02165	// -
OUTP      M13814	// T)R_3rd ROT Y SPANKING IN POS PLS
; L55
LOAD      M13814	// T)R_3rd ROT Y SPANKING IN POS PLS
AND NOT   M04161	// -
AND       T0716	// -
AND       P0008A	// -
AND       T1120	// R_4th FPCB SUPPORT UP
AND       P00085	// -
AND       P00087	// -
AND       P0005D	// R_P&P UP (SENSOR)
AND       M04140	// R_3rd SPK Y IN POS
OUTP      M13816	// T)R_3rd ROT Y SPANKING IN POS ->
// ======================== 18_R_3rd BENDING Z ==========================
; L57
LOAD      M02184	// T)R_3rd BD Z UP POS ->
OUTP      M1281A	// T)R_3rd BD Z UP POS ->
; L58
LOAD      M1281A	// T)R_3rd BD Z UP POS ->
OR        M12563	// R_1st MAND TOP CLAMP ORIGIN->
AND NOT   M04180	// R_3rd BD Z UP POS
AND       T0718	// R_3rd BD Z READY 2s
OUTP      M1281B	// T)R_3rd BD Z UP POS ->
; L60
LOAD      M02185	// T)R_3rd BD Z CENTER POS ->
OUTP      M1281C	// T)R_3rd BD Z CENTER POS ->
; L61
LOAD      M1281C	// T)R_3rd BD Z CENTER POS ->
AND NOT   M04181	// R_3rd BD Z CENTER POS
AND       T0718	// R_3rd BD Z READY 2s
AND       M04100	// R_P&P Y IDLE POS
OUTP      M1281D	// T)R_3rd BD Z CENTER POS ->
; L62
LOAD      M02186	// T)R_3rd BD Z BENDING POS ->
OUTP      M1281E	// T)R_3rd BD Z BENDING POS ->
; L63
LOAD      M1281E	// T)R_3rd BD Z BENDING POS ->
AND NOT   M04182	// R_3rd BD Z BENDING POS
AND       T0718	// R_3rd BD Z READY 2s
AND       M04100	// R_P&P Y IDLE POS
AND       T1085	// R_3rd DIE ALIGN BACKWARD
AND       T1086	// R_3rd DIE FPCB ALIGN BACKWARD
OUTP      M1281F	// T)R_3rd BD Z BENDING POS ->
; L64
MCSCLR    4

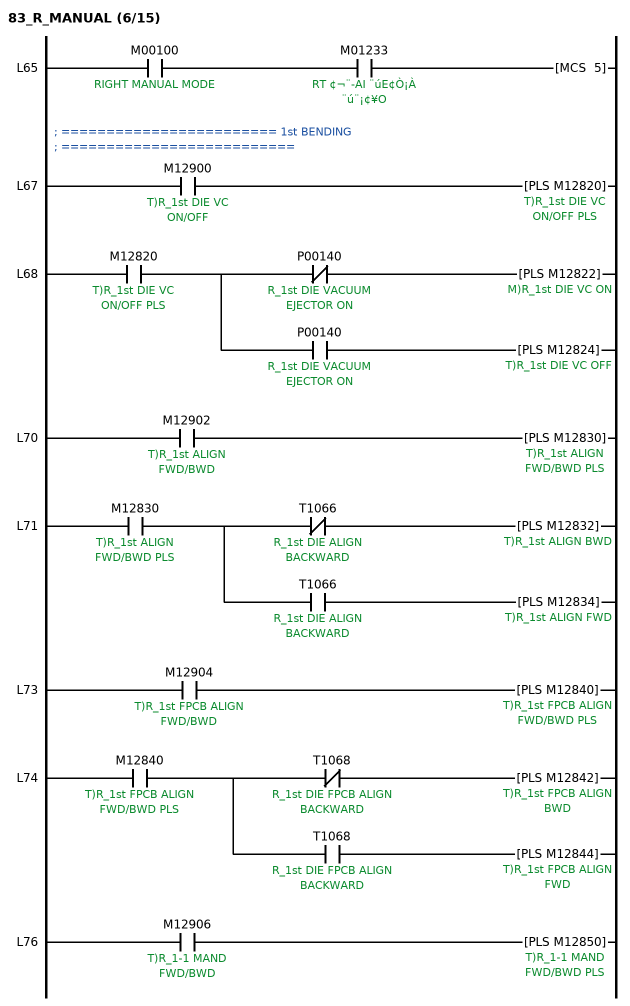
; L65
LOAD      M00100	// RIGHT MANUAL MODE
AND       M01233	// RT ¢¬¨­AI ¨úE¢Ò¡À ¨ú¨¡¢¥O
MCS       5
// ======================== 1st BENDING ==========================
; L67
LOAD      M12900	// T)R_1st DIE VC ON/OFF
OUTP      M12820	// T)R_1st DIE VC ON/OFF PLS
; L68
LOAD      M12820	// T)R_1st DIE VC ON/OFF PLS
MPUSH
AND NOT   P00140	// R_1st DIE VACUUM EJECTOR ON
OUTP      M12822	// M)R_1st DIE VC ON
MPOP
AND       P00140	// R_1st DIE VACUUM EJECTOR ON
OUTP      M12824	// T)R_1st DIE VC OFF
; L70
LOAD      M12902	// T)R_1st ALIGN FWD/BWD
OUTP      M12830	// T)R_1st ALIGN FWD/BWD PLS
; L71
LOAD      M12830	// T)R_1st ALIGN FWD/BWD PLS
MPUSH
AND NOT   T1066	// R_1st DIE ALIGN BACKWARD
OUTP      M12832	// T)R_1st ALIGN BWD
MPOP
AND       T1066	// R_1st DIE ALIGN BACKWARD
OUTP      M12834	// T)R_1st ALIGN FWD
; L73
LOAD      M12904	// T)R_1st FPCB ALIGN FWD/BWD
OUTP      M12840	// T)R_1st FPCB ALIGN FWD/BWD PLS
; L74
LOAD      M12840	// T)R_1st FPCB ALIGN FWD/BWD PLS
MPUSH
AND NOT   T1068	// R_1st DIE FPCB ALIGN BACKWARD
OUTP      M12842	// T)R_1st FPCB ALIGN BWD
MPOP
AND       T1068	// R_1st DIE FPCB ALIGN BACKWARD
OUTP      M12844	// T)R_1st FPCB ALIGN FWD
; L76
LOAD      M12906	// T)R_1-1 MAND FWD/BWD
OUTP      M12850	// T)R_1-1 MAND FWD/BWD PLS

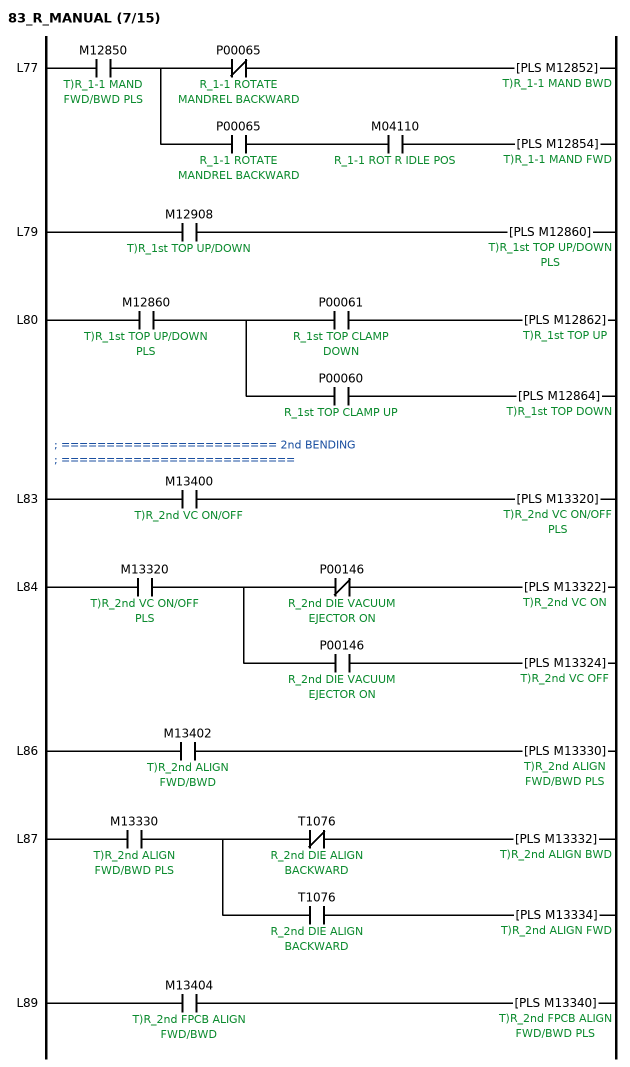
; L77
LOAD      M12850	// T)R_1-1 MAND FWD/BWD PLS
MPUSH
AND NOT   P00065	// R_1-1 ROTATE MANDREL BACKWARD
OUTP      M12852	// T)R_1-1 MAND BWD
MPOP
AND       P00065	// R_1-1 ROTATE MANDREL BACKWARD
AND       M04110	// R_1-1 ROT R IDLE POS
OUTP      M12854	// T)R_1-1 MAND FWD
; L79
LOAD      M12908	// T)R_1st TOP UP/DOWN
OUTP      M12860	// T)R_1st TOP UP/DOWN PLS
; L80
LOAD      M12860	// T)R_1st TOP UP/DOWN PLS
MPUSH
AND       P00061	// R_1st TOP CLAMP DOWN
OUTP      M12862	// T)R_1st TOP UP
MPOP
AND       P00060	// R_1st TOP CLAMP UP
OUTP      M12864	// T)R_1st TOP DOWN
// ======================== 2nd BENDING ==========================
; L83
LOAD      M13400	// T)R_2nd VC ON/OFF
OUTP      M13320	// T)R_2nd VC ON/OFF PLS
; L84
LOAD      M13320	// T)R_2nd VC ON/OFF PLS
MPUSH
AND NOT   P00146	// R_2nd DIE VACUUM EJECTOR ON
OUTP      M13322	// T)R_2nd VC ON
MPOP
AND       P00146	// R_2nd DIE VACUUM EJECTOR ON
OUTP      M13324	// T)R_2nd VC OFF
; L86
LOAD      M13402	// T)R_2nd ALIGN FWD/BWD
OUTP      M13330	// T)R_2nd ALIGN FWD/BWD PLS
; L87
LOAD      M13330	// T)R_2nd ALIGN FWD/BWD PLS
MPUSH
AND NOT   T1076	// R_2nd DIE ALIGN BACKWARD
OUTP      M13332	// T)R_2nd ALIGN BWD
MPOP
AND       T1076	// R_2nd DIE ALIGN BACKWARD
OUTP      M13334	// T)R_2nd ALIGN FWD
; L89
LOAD      M13404	// T)R_2nd FPCB ALIGN FWD/BWD
OUTP      M13340	// T)R_2nd FPCB ALIGN FWD/BWD PLS

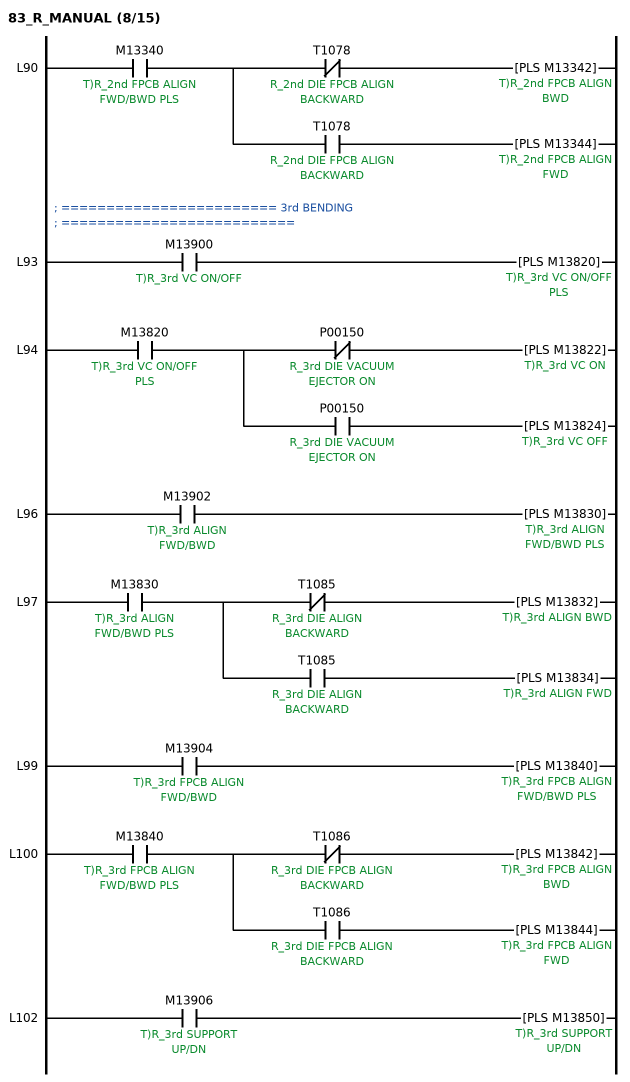
; L90
LOAD      M13340	// T)R_2nd FPCB ALIGN FWD/BWD PLS
MPUSH
AND NOT   T1078	// R_2nd DIE FPCB ALIGN BACKWARD
OUTP      M13342	// T)R_2nd FPCB ALIGN BWD
MPOP
AND       T1078	// R_2nd DIE FPCB ALIGN BACKWARD
OUTP      M13344	// T)R_2nd FPCB ALIGN FWD
// ======================== 3rd BENDING ==========================
; L93
LOAD      M13900	// T)R_3rd VC ON/OFF
OUTP      M13820	// T)R_3rd VC ON/OFF PLS
; L94
LOAD      M13820	// T)R_3rd VC ON/OFF PLS
MPUSH
AND NOT   P00150	// R_3rd DIE VACUUM EJECTOR ON
OUTP      M13822	// T)R_3rd VC ON
MPOP
AND       P00150	// R_3rd DIE VACUUM EJECTOR ON
OUTP      M13824	// T)R_3rd VC OFF
; L96
LOAD      M13902	// T)R_3rd ALIGN FWD/BWD
OUTP      M13830	// T)R_3rd ALIGN FWD/BWD PLS
; L97
LOAD      M13830	// T)R_3rd ALIGN FWD/BWD PLS
MPUSH
AND NOT   T1085	// R_3rd DIE ALIGN BACKWARD
OUTP      M13832	// T)R_3rd ALIGN BWD
MPOP
AND       T1085	// R_3rd DIE ALIGN BACKWARD
OUTP      M13834	// T)R_3rd ALIGN FWD
; L99
LOAD      M13904	// T)R_3rd FPCB ALIGN FWD/BWD
OUTP      M13840	// T)R_3rd FPCB ALIGN FWD/BWD PLS
; L100
LOAD      M13840	// T)R_3rd FPCB ALIGN FWD/BWD PLS
MPUSH
AND NOT   T1086	// R_3rd DIE FPCB ALIGN BACKWARD
OUTP      M13842	// T)R_3rd FPCB ALIGN BWD
MPOP
AND       T1086	// R_3rd DIE FPCB ALIGN BACKWARD
OUTP      M13844	// T)R_3rd FPCB ALIGN FWD
; L102
LOAD      M13906	// T)R_3rd SUPPORT UP/DN
OUTP      M13850	// T)R_3rd SUPPORT UP/DN

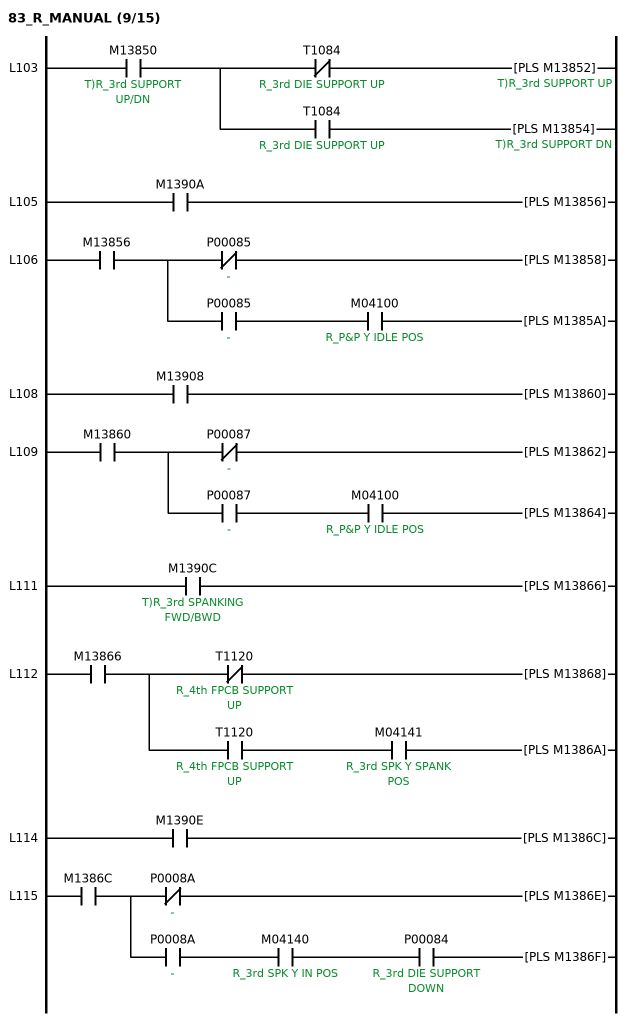
; L103
LOAD      M13850	// T)R_3rd SUPPORT UP/DN
MPUSH
AND NOT   T1084	// R_3rd DIE SUPPORT UP
OUTP      M13852	// T)R_3rd SUPPORT UP
MPOP
AND       T1084	// R_3rd DIE SUPPORT UP
OUTP      M13854	// T)R_3rd SUPPORT DN
; L105
LOAD      M1390A
OUTP      M13856
; L106
LOAD      M13856
MPUSH
AND NOT   P00085	// -
OUTP      M13858
MPOP
AND       P00085	// -
AND       M04100	// R_P&P Y IDLE POS
OUTP      M1385A
; L108
LOAD      M13908
OUTP      M13860
; L109
LOAD      M13860
MPUSH
AND NOT   P00087	// -
OUTP      M13862
MPOP
AND       P00087	// -
AND       M04100	// R_P&P Y IDLE POS
OUTP      M13864
; L111
LOAD      M1390C	// T)R_3rd SPANKING FWD/BWD
OUTP      M13866
; L112
LOAD      M13866
MPUSH
AND NOT   T1120	// R_4th FPCB SUPPORT UP
OUTP      M13868
MPOP
AND       T1120	// R_4th FPCB SUPPORT UP
AND       M04141	// R_3rd SPK Y SPANK POS
OUTP      M1386A
; L114
LOAD      M1390E
OUTP      M1386C
; L115
LOAD      M1386C
MPUSH
AND NOT   P0008A	// -
OUTP      M1386E
MPOP
AND       P0008A	// -
AND       M04140	// R_3rd SPK Y IN POS
AND       P00084	// R_3rd DIE SUPPORT DOWN
OUTP      M1386F

